# B&R Automation Studio project MotionTestBenchMaster (part 14)

### HMI_ICO.typ
```iecst
TYPE
	HMI_ICO_Type : 	STRUCT
		NextRecipeId : UDINT; (*ID of the next recipe requested from HLI*)
		ActualRecipeId : UDINT; (*ID of the actual recipe*)
		NextRecipeLoadingReq : BOOL; (*Request to download the new recipe*)
		RecipeLoaded : BOOL; (*New recipe downloaded*)
	END_STRUCT;
END_TYPE
```

### HMI_ITC.typ
```iecst
TYPE
	HMI_MachineComm_Type : 	STRUCT
		CapFault : BOOL; (*V4.A.A.1.6.12*)
		SkidFault : BOOL;
		FmcFault : BOOL;
	END_STRUCT;
END_TYPE
```

### HMI_MAU.typ
```iecst
(*DBA glass Status*)

TYPE
	HMI_DMC_Status : 	STRUCT
		Sector1Position : USINT;
		Sector1PistonDown : USINT;
		Sector1RotationToProd : USINT;
		Sector1RotationToCip : USINT;
		Sector1PistonUp : USINT;
		Sector2Position : USINT;
		Sector2PistonDown : USINT;
		Sector2RotationToProd : USINT;
		Sector2RotationToCip : USINT;
		Sector2PistonUp : USINT;
	END_STRUCT;
END_TYPE

(*COMMON*)

TYPE
	HMI_UV_Lamp_Type : 	STRUCT
		ConfigPresent : USINT;
		On : USINT;
		Ready : USINT;
		Alarm : USINT;
	END_STRUCT;
END_TYPE

(*GREASING*)

TYPE
	HMI_GrLb_Data_Type : 	STRUCT
		Alarm : BOOL;
		Pause : UINT; (*[laps]*)
		CycleTimeOut : UINT; (*[s]*)
		CycleNr : UINT; (*[#]*)
	END_STRUCT;
END_TYPE

(*SAFE LOGIC*)

TYPE
	HMI_SL_Info_Type : 	STRUCT
		RemoteCtrlStatus : UINT;
		CRC : UDINT;
		Password : ARRAY[0..15]OF USINT;
		Date : STRING[15];
		Author : STRING[32];
		IDMissed : STRING[80];
		IDMismatches : STRING[80];
		IDDiffFirmware : STRING[80];
		Led : HMI_SL_Led_Type;
	END_STRUCT;
	HMI_SL_Led_Type : 	STRUCT
		FAIL : USINT;
		FW_ACKN : USINT;
		MXCHG : USINT;
		RE : USINT;
	END_STRUCT;
	HMI_SL_PB_Type : 	STRUCT
		Ack_SK : PB_Type;
		Ack1UdId : PB_Type;
		Ack2UdId : PB_Type;
		Ack3UdId : PB_Type;
		Ack4UdId : PB_Type;
		AckMore4UdId : PB_Type;
		AckFW : PB_Type;
		LedTest : PB_Type;
		Scan : PB_Type;
	END_STRUCT;
	HMI_MAU_ChlRns_Type : 	STRUCT  (*master nuovo*)
		AVE260_PauseTimeWithBottles : UINT;
		AVE260_WorkTimeWithBottles : UINT;
		AVE260_PauseTimeWithoutBottles : UINT;
		AVE260_WorkTimeWithoutBottles : UINT;
		AVE261_PauseTimeWithoutBottles : UINT;
		AVE261_WorkTimeWithoutBottles : UINT;
		PauseTimeMaxWithoutChlRns : UINT;
		WorkTimeMaxWithoutChlRns : UINT;
	END_STRUCT;
END_TYPE
```

### HMI_MC.typ
```iecst
TYPE
	ST_HmiNewAxisData : 	STRUCT  (*V4.A.A.1.7.0*)
		rTorque : REAL;
		rTotalPhasingOffset : REAL;
		rMaxTorque : REAL;
		rPosition : REAL;
		rPosition_mm : REAL;
		rVelocity : REAL;
		rMotorTemperature : REAL;
		rLagError : REAL;
		rEncoderTemperature : REAL;
		rSwitchValue : REAL;
		rPrevAx_Position_mm : REAL;
		rHomingOffset : REAL; (*mm*)
		rNextAx_Position_mm : REAL;
		usiHmiName : USINT;
		uiDiagCode : UINT;
		uiAxisID : UINT; (*//Hmi Test*)
		iPrevAx_Number : INT;
		iNextAx_Number : INT;
		xMotorWithBrake : BOOL;
		xVelocityControl : BOOL;
		xInduction : BOOL;
		xReal : BOOL;
		xInitialized : BOOL;
		xEnabled : BOOL;
		xPowered : BOOL;
		xHomed : BOOL;
		xActive : BOOL;
		xInPosition : BOOL;
		xRunning : BOOL;
		xSynchro : BOOL;
		xBrakeReleased : BOOL;
		xFollowingError : BOOL;
		xInError : BOOL;
		xTorqueError : BOOL;
		xThirdPartMotor : BOOL;
		xHmiPresent : BOOL; (*//Hmi Test*)
		xHmiWait : BOOL;
	END_STRUCT;
	ST_HmiAxisData : 	STRUCT
		rTorque : REAL;
		rTotalPhasingOffset : REAL;
		rMaxTorque : REAL;
		rPosition : REAL;
		rPosition_mm : REAL;
		rVelocity : REAL;
		rMotorTemperature : REAL;
		rLagError : REAL;
		rEncoderTemperature : REAL;
		rSwitchValue : REAL;
		rPrevAx_Position_mm : REAL;
		rHomingOffset : REAL; (*mm*)
		rNextAx_Position_mm : REAL;
		usiHmiName : USINT;
		uiDiagCode : UINT;
		iPrevAx_Number : INT;
		iNextAx_Number : INT;
		xMotorWithBrake : BOOL;
		xVelocityControl : BOOL;
		xInduction : BOOL;
		xReal : BOOL;
		xInitialized : BOOL;
		xEnabled : BOOL;
		xPowered : BOOL;
		xHomed : BOOL;
		xActive : BOOL;
		xInPosition : BOOL;
		xRunning : BOOL;
		xSynchro : BOOL;
		xBrakeReleased : BOOL;
		xFollowingError : BOOL;
		xInError : BOOL;
		xTorqueError : BOOL;
		xThirdPartMotor : BOOL;
		xHmiWait : BOOL;
	END_STRUCT;
	ST_HmiMachineStatus : 	STRUCT
		xNoOperationActive : BOOL;
		xAuto : BOOL;
		xAutoCombi : BOOL;
		xPositioning : BOOL;
		xJogMachine : BOOL;
		xBrakeRelease : BOOL;
		xStepByStep : BOOL;
		xEndlessFeed : BOOL;
		xSplittedModality : BOOL;
		xFillerJogStandAlone : BOOL;
		xOutletJogStandAlone : BOOL;
		xInletJogStandAlone : BOOL;
		xFillerStepByStep : BOOL;
		xOutletStepByStep : BOOL;
		xInletStepByStep : BOOL;
		xFillerSlowMotion : BOOL;
		xOutletSlowMotion : BOOL;
		xInletSlowMotion : BOOL;
		xMachineStart : BOOL;
		xMachineSincroStop : BOOL;
		xMachineFixedSpeed : BOOL;
		xMachineSincro : BOOL;
		xMachineSincroInProgress : BOOL;
		xMachineOnError : BOOL;
		xMachineHomed : BOOL;
		xMachineRunning : BOOL;
		rEncoderPosition : REAL;
		rMachineStep : REAL;
	END_STRUCT;
	ST_HmiAxisPresent : 	STRUCT
		_99 : UINT;
		_100 : UINT;
		_105 : UINT;
		_106 : UINT;
		_107 : UINT;
		_108 : UINT;
		_109 : UINT;
		_110 : UINT;
		_111 : UINT;
		_112 : UINT;
		_113 : UINT;
		_114 : UINT;
		_115 : UINT;
		_116 : UINT;
		_117 : UINT;
		_118 : UINT;
		_119 : UINT;
		_120 : UINT;
		_121 : UINT;
		_200 : UINT;
		_211 : UINT;
		_212 : UINT;
		_213 : UINT;
		_214 : UINT;
		_215 : UINT;
		_216 : UINT;
		_217 : UINT;
		_218 : UINT;
		_219 : UINT;
		_300 : UINT;
		_311 : UINT;
		_312 : UINT;
		_313 : UINT;
		_314 : UINT;
		_315 : UINT;
		_316 : UINT;
		_317 : UINT;
		_318 : UINT;
		_319 : UINT;
	END_STRUCT;
	ST_HMIEncoderDiagnostic : 	STRUCT
		Present : BOOL;
		ModuleOK : BOOL;
		Value : DINT;
	END_STRUCT;
END_TYPE
```

### HMI_MNM.typ
```iecst
TYPE
	HMI_SpeedWidget_Type : 	STRUCT
		Modality : BOOL; (*0 = Auto / 1 = Jog*)
		Visibility : BOOL; (*0 = Hidden (Combi Mode) / 1 = Visible*)
		ActualSpeed : DINT; (*Actual Machine Speed [cph]*)
		AutoSpeedReq : DINT; (*Automatic Speed Required (Standalone) [cph]*)
		JogSpeedReq : DINT; (*Jog Speed Required (Standalone) [cph]*)
		Status : USINT; (*0: Error
1: Automatic
2: Jog
3: Adjustement
4: Slow motion forward
5: Slow motion backward*)
	END_STRUCT;
END_TYPE
```

### HMI_MNT.typ
```iecst
TYPE
	HMI_MNT_Type : 	STRUCT
		Macao : HMI_Macao_Type;
		Tpm : ARRAY[0..12]OF HMI_Tpm_Type; (*//v1.5*)
		_201QTB : HMI_Tpm_Type; (*V1.7.4*)
		_202QTB : HMI_Tpm_Type; (*V1.7.4*)
	END_STRUCT;
	HMI_Macao_Type : 	STRUCT
		Counter : ARRAY[0..15]OF UDINT;
		Event : ARRAY[0..7]OF BOOL;
	END_STRUCT;
	HMI_Tpm_Type : 	STRUCT  (*//v1.5*)
		Config : BOOL;
		AnalogNomValueVisible : BOOL;
		AnalogAlarmValueVisible : BOOL; (*V1.7.4*)
		InstrumentFault : BOOL; (*V1.7.4*)
		HmiID : UINT;
		AnalogActValue : REAL;
		AnalogMaxValue : REAL;
		AnalogMinValue : REAL;
		AnalogNomValue : REAL;
		AnalogAlarmValue : REAL; (*V1.7.4*)
	END_STRUCT;
END_TYPE
```

### HMI_OPS.typ
```iecst
TYPE
	HMI_OPS_Zone_Type : 	STRUCT
		Closed : BOOL;
		Locked : BOOL;
		LockSafety : BOOL;
		ShortSafety : BOOL;
		UnlockCommand : BOOL;
		Unlocked : BOOL;
		UnlockEnable : BOOL;
		UnlockRequest : BOOL;
		UnlockSafety : BOOL;
	END_STRUCT;
	HMI_OPS_Door_Type : 	STRUCT
		Confirm : BOOL;
		Lock1oo2 : BOOL;
		LockSafety : BOOL;
		Opened : BOOL;
		ShortCircuit : BOOL;
		UnLock : BOOL;
	END_STRUCT;
	HMI_OPS_Emergency_Type : 	STRUCT
		I_Pressed : BOOL;
		I_short_Fault : BOOL;
	END_STRUCT;
	HMI_OPS_Jog_Type : 	STRUCT
		ShCircPlug : BOOL;
		ShCircStop : BOOL;
		Stop : BOOL;
		Plugged : BOOL;
	END_STRUCT;
	HMI_SafetyWidget_Type : 	STRUCT
		ZoneAlarm : ARRAY[MIN_CFG_SafetyZone..MAX_CFG_SafetyZone]OF BOOL;
		BufferAlarm : BOOL;
	END_STRUCT;
	HMI_OPS_Pictogram_Type : 	STRUCT
		AccesOk : BOOL;
		AccesReq : BOOL;
		Acces : BOOL;
		Chemical : BOOL;
		Temperature : BOOL;
	END_STRUCT;
	HMI_OPS_RfidAccess_Type : 	STRUCT
		Present : BOOL; (*Module Present*)
		CodeFault : BOOL; (*Code discrepancy*)
		KeyFault : BOOL; (*Key not recognised*)
		KeyOk : BOOL; (*Key present and recognised*)
	END_STRUCT;
	HMI_OPS_SafetySwitch_Type : 	STRUCT  (*V4.A.A.1.7.1*) (* *) (*139*)
		ShortFault : BOOL; (*Short circuit fault on PB*) (* *) (*141*)
		SwitchOn : BOOL; (*Switch active*) (* *) (*143*)
		Visibility : BOOL; (*Switch present*) (* *) (*144*)
	END_STRUCT;
END_TYPE
```

### HMI_RNS.typ
```iecst
TYPE
	HMI_RNS_ManualCapsSelection_Type : 	STRUCT  (*V4.A.A.1.7.0*)
		Value : USINT;
		Visibility : BOOL;
	END_STRUCT;
	HMI_RNS_State_Type : 	STRUCT (*V4.A.A.1.7.4*)
		Sequencer : Seq_Type; (*Step Actual*)
		Signals : Signals_Type;
	END_STRUCT;
END_TYPE
```

### HMI_SFT.typ
```iecst
TYPE
	StepAcquisition_Type : 	STRUCT
		Step : USINT;
		_207DSF : StepAcquisition_Sensor_Type;
		_208DSF : StepAcquisition_Sensor_Type;
		_202DSF : StepAcquisition_Sensor_Type;
		_203DSF : StepAcquisition_Sensor_Type;
	END_STRUCT;
	StepAcquisition_Sensor_Type : 	STRUCT
		Visibility : BOOL;
		Value : UINT;
	END_STRUCT;
	MainCounters_Type : 	STRUCT
		PbResetMachineCounters : PB_Type;
		MachineCounters : MachineCounters_Type;
		PbResetCycleCounters : PB_Type;
		CycleCounters : TankCounters_Type;
		PbResetContainersCounters : PB_Type;
		ContainersCounters : ContainersCounters_Type;
		PbResetEcoEitCounters : PB_Type;
		EcoEitCounters : EcoEitCounters_Type;
	END_STRUCT;
	MachineCounters_Type : 	STRUCT
		CapLaps : UDINT; (*Capper torret laps counter*)
		FlrLaps : UDINT; (*Filler laps counter*)
		RnsLaps : UDINT; (*Rinser laps counter*)
		PowerOnCycles : UDINT;
		PowerOnTime : CounterTime_Type;
		RotationTime : CounterTime_Type; (*Machine running hours counter*)
		StartTime : CounterTime_Type;
	END_STRUCT;
	ContainersCounters_Type : 	STRUCT
		CapFault : UDINT;
		FlrBurst : UDINT;
		RnsFault : UDINT;
		FlrFault : UDINT;
		Ejected : UDINT;
		Entered : UDINT;
		Produced : UDINT;
		StartTime : CounterTime_Type;
	END_STRUCT;
	TankCounters_Type : 	STRUCT
		ProductionCounter : UDINT;
		ProductionTime : CounterTime_Type;
		CipCounter : UDINT;
		CipTime : CounterTime_Type;
		StartTime : CounterTime_Type;
	END_STRUCT;
	EcoEitCounters_Type : 	STRUCT
		ElectricalPowerKWH : REAL; (*[KWH]*)
		ElectricalPowerKVAR : REAL; (*[KVAR]*)
		StartTime : CounterTime_Type;
	END_STRUCT;
	HmiCounterData_Type : 	STRUCT
		Description : STRING[25];
		Unit : STRING[8];
		PbReset : PB_Type;
		ConfigPresent : BOOL;
		ValuePresent : BOOL;
		TimePresent : BOOL;
		StartDatePresent : BOOL;
	END_STRUCT;
	CounterCfg_Type : 	STRUCT
		MachineCounters : MachineCountersCfg_Type;
		ContainersCounters : ContainersCountersCfg_Type;
		ProcessCounters : ProcessCountersCfg_Type;
		EcoCounters : EcoCountersCfg_Type;
	END_STRUCT;
	CounterData_Type : 	STRUCT
		MachineCounters : MachineCountersData_Type;
		ContainersCounters : ContainersCountersData_Type;
		ProcessCounters : ProcessCountersData_Type;
		EcoCounters : EcoCountersData_Type;
	END_STRUCT;
	HMI_CounterPage_Type : 	STRUCT
		Partial : HMI_CounterPage2_Type;
		Total : HMI_CounterPage2_Type;
	END_STRUCT;
	HMI_CounterPage2_Type : 	STRUCT
		Data : ARRAY[0..15]OF HmiCounterData_Type;
		Cfg : ARRAY[0..15]OF Counters_Type;
	END_STRUCT;
END_TYPE

(*Machine Counter*)

TYPE
	MachineCountersCfg_Type : 	STRUCT
		HmiData : ARRAY[0..15]OF HmiCounterData_Type;
	END_STRUCT;
	MachineCountersData_Type : 	STRUCT
		CounterData : ARRAY[0..15]OF Counters_Type;
	END_STRUCT;
END_TYPE

(*Containers Counter*)

TYPE
	ContainersCountersCfg_Type : 	STRUCT
		HmiData : ARRAY[0..15]OF HmiCounterData_Type;
	END_STRUCT;
	ContainersCountersData_Type : 	STRUCT
		CounterData : ARRAY[0..15]OF Counters_Type;
	END_STRUCT;
END_TYPE

(*Process Coutner*)

TYPE
	ProcessCountersCfg_Type : 	STRUCT
		HmiData : ARRAY[0..15]OF HmiCounterData_Type;
	END_STRUCT;
	ProcessCountersData_Type : 	STRUCT
		CounterData : ARRAY[0..15]OF Counters_Type;
	END_STRUCT;
END_TYPE

(*Eco Counter*)

TYPE
	EcoCountersCfg_Type : 	STRUCT
		HmiData : ARRAY[0..15]OF HmiCounterData_Type;
	END_STRUCT;
	EcoCountersData_Type : 	STRUCT
		CounterData : ARRAY[0..15]OF Counters_Type;
	END_STRUCT;
END_TYPE

(*FILLING VALVE*)

TYPE
	DummyContainerDataStructure_Type : 	STRUCT
		FillingNozzle : USINT;
		DummyInstalled : BOOL; (*SHIFT master nuovo*)
		DummyNotInserted : BOOL;
		DummyRemoved : BOOL;
		DummyNotRemoved : BOOL;
	END_STRUCT;
	FillingValveDataStructure_Type : 	STRUCT
		FillingDisabled : BOOL; (*SHIFT master nuovo*)
		ContainerBurst : BOOL;
		ContainerPresence : BOOL;
		PreClosingEnd : BOOL;
		WashingLapsEnd : BOOL;
		PreClosingCmdLap1 : BOOL;
		PreClosingCmdLap2 : BOOL;
		PreClosingCmdLap3 : BOOL;
		PreClosingCmdLap4 : BOOL;
		PreClosingCmdLap5 : BOOL;
		PreClosingCmdLap6 : BOOL;
		PreClosingCmdLap7 : BOOL;
		OperatorInspectionReq : BOOL;
		PreClosingActualLap : USINT;
		WashingLaps : USINT;
		ConsecutiveFillNotOk : USINT;
		AbsoluteFillNotOk : USINT;
		ConsecutiveBurst : USINT;
		AbsoluteBurst : USINT;
	END_STRUCT;
	HMI_SFT_BurstData_Type : 	STRUCT
		ColorStatus : USINT;
		Counter : UINT;
	END_STRUCT;
END_TYPE

(*Sampling*)

TYPE
	HMI_SFT_SamplingMold_Type : 	STRUCT  (*V1.61*)
		Present : BOOL;
		Selected : BOOL;
	END_STRUCT;
END_TYPE
```

### HMI.typ
```iecst
TYPE
	Step_Type : 	STRUCT
		Config_Visualization : BOOL;
		Preset : REAL; (*Preset Step Time*)
		Actual : REAL; (*Actual Step Time*)
		StepIndex : UINT; (*Actual Sequencer Step Number*)
		StepIndexText : UINT; (*Request Step Text to HMI*)
	END_STRUCT;
	Signals_Type : 	STRUCT
		DigitalIn : ARRAY[1..5]OF HMI_DigitalITC_Type;
		AnalogIn : ARRAY[1..2]OF HMI_AnalogITC_Type;
		DigitalOut : ARRAY[1..5]OF HMI_DigitalITC_Type;
		AnalogOut : ARRAY[1..2]OF HMI_AnalogITC_Type;
	END_STRUCT;
	Seq_Type : 	STRUCT
		TextBar : ARRAY[0..4]OF SeqTextBar_Type;(*master nuovo*)
		InfoBox : ARRAY[0..5]OF SeqInfo_Type; (*Preset Step Time*)
	END_STRUCT;
	SeqTextBar_Type : 	STRUCT
		Visibility : BOOL;
		IndexNr : UINT; (*Actual Sequencer Step Number*)
		IndexText : UINT; (*Request Step Text to HMI*)
	END_STRUCT;
	SeqInfo_Type : 	STRUCT
		Visibility : BOOL;
		IndexText : STRING[20]; (*Request Step Text to HMI*)
		Unit : UINT;
		ProgressVisibility : BOOL; (*Step Progress Visibility*)
		Progress : REAL; (*Step Progress Time*)
		Preset : REAL; (*Preset Step Time*)
		Actual : REAL; (*Actual Step Time*)
	END_STRUCT;
	Info_Type : 	STRUCT  (*v1.4*)
		Visibility : BOOL;
		Preset : REAL; (*Preset Value*)
		Actual : REAL; (*Actual value*)
	END_STRUCT;
	Data_Type : 	STRUCT  (*v1.7.4a*)
		Visibility : BOOL;
		StringLineNameVisibility : BOOL; (*0=Fix text displayed-1= String displayed*)
		DataValueVisibility : BOOL; (*0=String displayed-1= Numeric value displayed*)
		LineName : STRING[100]; (*Line Name*)
		DataText : STRING[100]; (*Data Text in Case of String*)
		DataValue : REAL; (*Data Value in Case of Numeric*)
	END_STRUCT;
	HMI_CounterHome_Type : 	STRUCT  (*V4.A.A.1.6.8*)
		SS2P : SS2P_Type;
		CounterValue : ARRAY[0..1]OF UDINT;
	END_STRUCT;
END_TYPE
```

### HMI_BTC.typ - not listed in the package file held
```iecst
(*BOTTLE BOTTOM COOLING*)

TYPE
	HMI_BTC_State_Type : 	STRUCT
		Sequencer : Seq_Type; (*Step Actual*)
		Signals : Signals_Type;
	END_STRUCT;
END_TYPE
```

### Package Logical/02_HMI/HMI_Variables - HMI Global variables

### HMI_AID.var
```iecst
VAR
	HMI_CmdBar_PB : ARRAY[MIN_CmdBar_PB..MAX_CmdBar_PB] OF CmdBarPB_Type := [25((Enable:=FALSE,LampON:=FALSE,Blink:=FALSE,Visibility:=FALSE,ON:=FALSE,Command:=FALSE))]; (*1: Mixer Start/Stop
2: Filler Start/Stop
3: Labeller Start/Stop
4: Blower Start/Stop
5: Labeller Master/Slave
6: Preform Loading
7: Bottle with label ejection
8: Empty bottle ejection
9: Preform ejection
10: Filler/Labeller coupling
11: Labeller/Blower coupling
12: Filler door unlock
13: Labeller door unlock
14: Blower door unlock*)
	HMI_PB : ARRAY[MIN_PB_CFG..MAX_PB_CFG] OF PB_Type;
	HMI_SS2P : ARRAY[MIN_SS2P_CFG..MAX_SS2P_CFG] OF SS2P_Type;
	HMI_SS2P_Custom : ARRAY[0..2] OF SS2PCustom_Type; (*V4.A.A.1.6.13*)
END_VAR
```

### HMI_ALR.var
```iecst
VAR
	HMI_ALR : ARRAY[1..8000] OF BYTE;
	HMI_MSG : ARRAY[1..2000] OF BOOL;
END_VAR
```

### HMI_CAP.var
```iecst
VAR
	HMI_CAP_Step : INT;
	HMI_CAP_PB : ARRAY[MIN_PB_CFG..MAX_PB_CFG] OF PB_Type;
	HMI_CAP_SS2P : ARRAY[MIN_SS2P_CFG..MAX_SS2P_CFG] OF SS2P_Type;
	HMI_CAP_SS3P : ARRAY[MIN_SS3P_CFG..MAX_SS3P_CFG] OF SS3P_Type;
	HMI_CAP_CapsTypeCFG : STRING[500];
	HMI_CAP_ManualCapsSelection : HMI_CAP_ManualCapsSelection_Type;
	HMI_CAP_State : HMI_CAP_State_Type;
	HMI_CAP_ConfigStructure : HMI_CAP_ConfigStructure_Type;
	HMI_CAP_BufferPresent : BOOL; (*Buffer Present bit for HMI*)
	HMI_CAP_MultiChoiceMng : USINT; (*1=Arol Equatorque ; 2=Arol Equatorque\Multybody ; 3=Zalkin Brushless ; 4=Siko Multybody*)
	HMI_CAP_Brush : HMI_CAP_Brush_Type; (*Capper Brushless Arol/Zalkin v1.4*)
	HMI_CAP_DataCfg : ARRAY[1..10] OF HMI_COP_ZoneCfg_Type; (*Column Configuration Capper Brushless Arol/Zalkin v1.4*)
	HMI_CAP_BufferAdjust : Info_Type; (*//V4.A.A.1.6.11*)
	HMI_CAP_HRM : HMI_CAP_HRM_Type; (*//V4.A.A.1.6.11*)
END_VAR
(*GREASING*)
VAR
	HMI_CAP_GreasingState : Seq_Type;
	HMI_CAP_GreasingState2 : Seq_Type; (*//V4.A.A.1.6.11*)
	HMI_CAP_GreasingData2 : HMI_CAP_Greasing_Type; (*//V4.A.A.1.6.11*)
	HMI_CAP_GreasingData : HMI_CAP_Greasing_Type;
END_VAR
(*MOTORS*)
VAR
	HMI_202GPE : HMI_GreasingPump_Type;
	HMI_203GPE : HMI_GreasingPump_Type; (*//V4.A.A.1.6.11*)
	HMI_206MMR : HMI_Motor_FC_Type; (*Head rotation motor*)
	HMI_206MMRBrake : HMI_Motor_Type; (*Head rotation motor*)
	HMI_207MMR : HMI_Motor_FC_Type; (*Hopper motor chute 1*)
	HMI_230MMR : HMI_Motor_Type; (*Dust removal motor on caps channel*)
	HMI_231MMR : HMI_Motor_Type; (*Dust removal motor on buffer //V4.A.A.1.6.11*)
	HMI_229MMR : HMI_Motor_Type; (*Adjustment panel motor //V4.A.A.1.6.11*)
	HMI_212MMR : HMI_Motor_FC_Type; (*Buffer rotation motor*)
	HMI_213MMR : HMI_Motor_Type; (*Head rotation motor fun*)
	HMI_214MMR : HMI_Motor_FC_Type; (*Hopper motor chute 2*)
	HMI_215MMR : HMI_Motor_FC_Type; (*Hopper motor chute 3*)
END_VAR
(*IONIZER*)
VAR
	HMI_201DRC_SwitchFeedback : HMI_DI_Type;
	HMI_201DRC : HMI_Motor_Type; (*Ionizer*)
END_VAR
(*UV LAMP*)
VAR
	HMI_201LLC : HMI_Motor_Type; (*UV lamp Chute 1*)
	HMI_202LLC : HMI_Motor_Type; (*UV lamp Chute 2*)
	HMI_203LLC : HMI_Motor_Type; (*UV lamp Chute 3*)
END_VAR
(*SIKO MULTIBODY V1.61*)
VAR
	HMI_CAP_SikoMotorSetPointEnable : BOOL; (*Multibody Siko Motor for Automatic Change Capper Guide Enable Set Point For Calibration*)
	HMI_CAP_SikoMotor : ARRAY[0..5] OF HMI_CAP_SikoMotor_Type; (*Multibody Siko Motor for Automatic Change Capper Guide *)
END_VAR
(*DRIVERS*)
VAR
	HMI_VFD_206MMR : HMI_Danfoss_Diag_Type; (*Head rotation motor*)
	HMI_VFD_207MMR : HMI_Danfoss_Diag_Type; (*Hopper motor chute 1*)
	HMI_VFD_230MMR : HMI_Danfoss_Diag_Type; (*Dust remover motor*)
	HMI_VFD_212MMR : HMI_Danfoss_Diag_Type; (*Buffer rotation motor*)
	HMI_VFD_213MMR : HMI_Danfoss_Diag_Type; (*Head rotation motor fun*)
	HMI_VFD_214MMR : HMI_Danfoss_Diag_Type; (*Hopper motor chute 2*)
	HMI_VFD_215MMR : HMI_Danfoss_Diag_Type; (*Hopper motor chute 3*)
	HMI_ST3B : HMI_Analog_IN_Type; (*Tempaerature sensor Equatorque motor//V4.A.A.1.6.12*)
	HMI_ST3A : HMI_Analog_IN_Type; (*Tempaerature sensor Equatorque motor//V4.A.A.1.6.12*)
END_VAR
(*VALVES*)
VAR
	HMI_201CPC : HMI_Valve_Type; (*EV chute 1 caps release*)
	HMI_202CPC : HMI_Valve_Type; (*EV chute 2 caps release*)
	HMI_205CPC : HMI_Valve_Type; (*EV caps block chute 1*)
	HMI_206CPC : HMI_Valve_Type; (*EV caps block chute 2*)
	HMI_207CPC : HMI_Valve_Type; (*EV cap discharge door*)
	HMI_212CPC : HMI_Valve_Type; (*EV open buffer discharge door*)
	HMI_213CPC : HMI_Valve_Type; (*EV buffer lifting*)
	HMI_214CPC : HMI_Valve_Type; (*EV buffer lock*)
	HMI_215CPC : HMI_Valve_Type; (*EV lock size change guide*)
	HMI_216CPC : HMI_Valve_Type; (*EV 3 size change guide*)
	HMI_217CPC : HMI_Valve_Type; (*EV 4 size change guide*)
	HMI_218CPC : HMI_Valve_Type; (*EV sport size change guide*)
	HMI_219CPC : HMI_Valve_Type; (*EV open channel discharge door*)
	HMI_220CPC : HMI_Valve_Type; (*FREE v1.7.6*)
	HMI_221CPC : HMI_Valve_Type; (*EV chute 3 caps release*)
	HMI_222CPC : HMI_Valve_Type; (*EV caps block chute 3*)
	HMI_223CPC : HMI_Valve_Type; (*EV buffer vibrator*)
	HMI_224CPC : HMI_Valve_Type; (*EV cam position*)
	HMI_225CPC : HMI_Valve_Type; (*EV cam locking*)
	HMI_226CPC : HMI_Valve_Type; (*EV opening door UV Lamp A V. 1.1*)
	HMI_227CPC : HMI_Valve_Type; (*EV  Block Caps Outlet Chute 1*)
	HMI_228CPC : HMI_Valve_Type; (*EV transfer Starwheel air soleniod valve DA VERIFICARE*)
	HMI_229CPC : HMI_Valve_Type; (*EV transfer Starwheel air soleniod valve DA VERIFICARE*)
	HMI_232CPC : HMI_Valve_Type; (*EV opening door UV Lamp B V. 1.1*)
	HMI_233CPC : HMI_Valve_Type;
	HMI_234CPC : HMI_Valve_Type; (*EV Caps Ejection Cap Feeder V4.A.A.1.6.12*)
	HMI_235CPC : HMI_Valve_Type; (*v1.7.4*)
	HMI_236CPC : HMI_Valve_Type; (*v1.7.4*)
	HMI_237CPC : HMI_Valve_Type; (*v1.7.4*)
	HMI_238CPC : HMI_Valve_Type; (*v1.7.4*)
	HMI_201EVC : HMI_Valve_Type; (*Air blowing for cap release 1 V1.6*)
	HMI_203EVC : HMI_Valve_Type; (*Air blowing for cap release 2 V1.6*)
	HMI_207EVC : HMI_Valve_Type; (*Air blowing for cap release 3 V1.6*)
	HMI_209EVC : HMI_Valve_Type; (*v1.7.4*)
	HMI_210EVC : HMI_Valve_Type; (*Air blowing for buffer emptying*)
	HMI_211EVC : HMI_Valve_Type; (*Buffer air blowing for caps release*)
	HMI_212EVC : HMI_Valve_Type; (*Air blowing for chute emptying*)
	HMI_213EVC : HMI_Valve_Type; (*Air blowing caps ionizer chute 1*)
	HMI_214EVC : HMI_Valve_Type; (*Air blowing caps ionizer chute 2*)
	HMI_215EVC : HMI_Valve_Type; (*Air blowing caps ionizer chute 3*)
	HMI_216EVC : HMI_Valve_Type; (*Air blowing for chute emptying by pep*)
	HMI_227EVC : HMI_Valve_Type; (*v1.7.4*)
	HMI_228EVC : HMI_Valve_Type; (*v1.7.4*)
	HMI_229EVC : HMI_Valve_Type; (*v1.7.4*)
	HMI_203EVF : HMI_Valve_Type; (*Air blowing caps (Drying)*)
	HMI_AVC : ARRAY[MIN_CFG_AVC..MAX_CFG_AVC] OF HMI_Valve_Type; (*Caps Treatment Valves V4.A.A.1.7.4*)
END_VAR
(*SENSOR*)
VAR
	HMI_201DSC : HMI_Photocell_Type; (*Caps/crowns release check*)
	HMI_202DSC : HMI_DI_Type; (*Low level caps/crowns presence chute 1*)
	HMI_204DSC : HMI_DI_Type; (*Head 1 sensor*)
	HMI_205DSC : HMI_DI_Type; (*Lack of caps (Quibuf infeed)*)
	HMI_210DSC : HMI_DI_Type; (*Cap Overturned hight Cap Feeder  V4.A.A.1.7.1*)
	HMI_211DSC : HMI_DI_Type; (*Cap Overturned low  Cap Feeder  V4.A.A.1.7.1*)
	HMI_216DSC : HMI_DI_Type; (*Low level caps/crowns presence chute 2*)
	HMI_217DSC : HMI_DI_Type; (*Low level caps/crowns presence chute 3*)
	HMI_218DSC : HMI_DI_Type; (*Upside down caps check chute 1 high*)
	HMI_219DSC : HMI_DI_Type; (*Upside down caps check chute 1 low*)
	HMI_220DSC : HMI_DI_Type; (*Upside down caps check chute 2 high*)
	HMI_221DSC : HMI_DI_Type; (*Upside down caps check chute 2 low*)
	HMI_222DSC : HMI_DI_Type; (*Upside down caps check chute 3 high*)
	HMI_223DSC : HMI_DI_Type; (*Upside down caps check chute 3 low*)
	HMI_224DSC : HMI_DI_Type; (*Ionizer pressure switch chute 1*)
	HMI_225DSC : HMI_DI_Type; (*Ionizer pressure switch chute 2*)
	HMI_226DSC : HMI_DI_Type; (*Ionizer pressure switch chute 3*)
	HMI_227DSC : HMI_DI_Type; (*Lubrication door sensor*)
	HMI_228DSC : HMI_DI_Type; (*Fixed part lubrication check*)
	HMI_229DSC : HMI_DI_Type; (*Rotating part lubrication check*)
	HMI_230DSC : HMI_DI_Type; (*Lubrication pipe inserted sensor*)
	HMI_231DSC : HMI_DI_Type; (*Turret cam position analog sensor*)
	HMI_232DSC : HMI_DI_Type; (*Caps buffer full*)
	HMI_233DSC : HMI_DI_Type; (*Caps channel discharge gate sensor*)
	HMI_234DSC : HMI_DI_Type; (*Lubrication phase sensor*)
	HMI_235DSC : HMI_DI_Type; (*Buffer in high position*)
	HMI_236DSC : HMI_DI_Type; (*Buffer in low position*)
	HMI_237DSC : HMI_DI_Type; (*Buffer lock inserted*)
	HMI_238DSC : HMI_DI_Type; (*Caps buffer max level chute 1*)
	HMI_239DSC : HMI_DI_Type; (*Caps buffer max level chute 2*)
	HMI_240DSC : HMI_DI_Type; (*Caps buffer max level chute 3*)
	HMI_241DSC : HMI_DI_Type; (*Hopper level chute 1*)
	HMI_242DSC : HMI_DI_Type; (*Hopper level chute 2*)
	HMI_243DSC : HMI_DI_Type; (*Hopper level chute 3*)
	HMI_244DSC : HMI_DI_Type; (*Max level caps/crowns chute 1*)
	HMI_245DSC : HMI_DI_Type; (*Max level caps/crowns chute 2*)
	HMI_246DSC : HMI_DI_Type; (*Max level caps/crowns chute 3*)
	HMI_247DSC : HMI_DI_Type; (*Medium level caps/crowns chute 1*)
	HMI_248DSC : HMI_DI_Type; (*Medium level caps/crowns chute 2*)
	HMI_249DSC : HMI_DI_Type; (*Medium level caps/crowns chute 3*)
	HMI_250DSC : HMI_DI_Type; (*Side door hopper sport*)
	HMI_251DSC : HMI_DI_Type; (*Top door hopper sport*)
	HMI_252DSC : HMI_DI_Type; (*Uv lamp door*)
	HMI_253DSC : HMI_DI_Type; (*Sensore carter posteriore*)
	HMI_254DSC : HMI_DI_Type; (*Sensore di fase per lubrificazione*)
	HMI_255DSC : HMI_DI_Type; (*Sensore di lubrificazione della parte fissa*)
	HMI_256DSC : HMI_DI_Type; (*Sensore di lubrificazione della parte rotante*)
	HMI_257DSC : HMI_DI_Type; (*Sensore di inserimento del raccordo di lubrificazione della parte rotante *)
	HMI_258DSC : HMI_DI_Type; (*Sensore carter superiore  //V4.A.A.1.6.11*)
	HMI_259DSC : HMI_DI_Type; (*Sensore di lubrificazione rotazione teste  //V4.A.A.1.6.11*)
	HMI_260DSC : HMI_DI_Type; (*Sensore di inserimento del raccordo di lubrificazione della parte rotante riduttore rotazione teste  //V4.A.A.1.6.11*)
	HMI_261DSC : HMI_DI_Type; (*Sensore limite minimo posizione pannello //V4.A.A.1.6.11*)
	HMI_262DSC : HMI_DI_Type; (*Sensore zero encoder //V4.A.A.1.6.11*)
	HMI_263DSC : HMI_DI_Type; (*Sensore limite massimo posizione pannello //V4.A.A.1.6.11*)
	HMI_264DSC : HMI_Photocell_Type; (*Caps/Crown release check on bottle//V4.A.A.1.6.12h*)
	HMI_266DSC : HMI_DI_Type; (*v1.7.4*)
	HMI_267DSC : HMI_DI_Type; (*v1.7.5*)
	HMI_268DSC : HMI_DI_Type; (*v1.7.5*)
	HMI_270DSC : HMI_DI_Type; (*Caps Belt Sensor  // v1.7.4*)
END_VAR
```

### HMI_RNS.var
```iecst
(*RINSER*)
VAR
	HMI_RNS_PB : ARRAY[MIN_PB_CFG..MAX_PB_CFG] OF PB_Type;
	HMI_RNS_SS2P : ARRAY[MIN_SS2P_CFG..MAX_SS2P_CFG] OF SS2P_Type;
	HMI_RNS_SS3P : ARRAY[MIN_SS3P_CFG..MAX_SS3P_CFG] OF SS3P_Type;
	HMI_RNS_MultiChoiceMng : USINT; (*0=Rinser Instant Data Not Present  1=Rinser Instant Data Present V4.A.A.1.7.0*)
	HMI_RNS_State : HMI_RNS_State_Type;
	HMI_RNS_NozzleData : ARRAY[1..15] OF RNS_NozzleData_Type; (*V4.A.A.1.7.0*)
	HMI_RNS_ManualSelection : HMI_RNS_ManualCapsSelection_Type; (*V4.A.A.1.7.0*)
	HMI_RNS_TypeCFG : STRING[500]; (*V4.A.A.1.7.0*)
	HMI_RNS_Treatments : ARRAY[0..19] OF HMI_ComboBoxElements_Type := [(Present:=TRUE,Name:='Full Treatment'),(Present:=TRUE,Name:='Water Only'),(Present:=TRUE,Name:='Air Only'),14((0)),10((0)),1((0)),2((0))]; (*V4.A.A.1.7.0*)
END_VAR
```

### HMI_CO.var
```iecst
VAR
	HMI_CO_SS2P : ARRAY[MIN_SS2P_CFG..MAX_SS2P_CFG] OF SS2P_Type;
	HMI_APCO_TypeOfChangeCFG : STRING[500];
	HMI_APCO_TypeOfChange : ARRAY[1..16] OF BOOL; (*V4.A.A.1.6.12*)
END_VAR
VAR RETAIN
	HMI_APCO : HMI_APCO_Type;
END_VAR
```

### HMI_COP.var
```iecst
VAR
	HMI_COP_StatusWidget : HMI_COP_StatusWidget_Type;
END_VAR
VAR RETAIN
	HMI_COP_PB : ARRAY[MIN_PB_CFG..MAX_PB_CFG] OF PB_Type;
	HMI_COP_SS2P : ARRAY[MIN_SS2P_CFG..MAX_SS2P_CFG] OF SS2P_Type;
	HMI_COP_SS3P : ARRAY[MIN_SS3P_CFG..MAX_SS3P_CFG] OF SS3P_Type;
END_VAR
VAR
	HMI_COP_RcpTemp : HMI_COP_Rcp_Type;
END_VAR
VAR RETAIN
	HMI_COP_RcpSelection : ARRAY[0..CST_COP_RcpMax] OF HMI_COP_RcpSelection_Type;
END_VAR
VAR
	HMI_COP_RcpInfo : HMI_COP_RcpInfo_Type;
	HMI_COP_ZoneCfg : ARRAY[1..32] OF HMI_COP_ZoneCfg_Type;
END_VAR
VAR RETAIN
	HMI_RCP_COP_Mngt : RCP_Management_Type;
	HMI_COP_Rcp : HMI_COP_Rcp_Type;
END_VAR
VAR
	HMI_COP_State : HMI_COP_State_Type;
	HMI_COP_PhaseTypeCFG : STRING[500];
	HMI_COP_FuTypeCFG : UDINT;
	HMI_COP_FuGunTypeCFG : UDINT;
	HMI_COP_FuDrainableCFG : UDINT;
	HMI_COP_ITC : HMI_COP_ITC_Type;
	HMI_COP_OptPlangerPresent : BOOL; (*vrma*)
END_VAR
VAR RETAIN
	HMI_RCP_COP_SelectedRecipeName : STRING[70]; (*v999hema*)
END_VAR
```

### HMI_CRW.var
```iecst
VAR
	HMI_CRW_Step : INT;
	HMI_CRW_PB : ARRAY[MIN_PB_CFG..MAX_PB_CFG] OF PB_Type;
	HMI_CRW_SS2P : ARRAY[MIN_SS2P_CFG..MAX_SS2P_CFG] OF SS2P_Type;
	HMI_CRW_SS3P : ARRAY[MIN_SS3P_CFG..MAX_SS3P_CFG] OF SS3P_Type;
	HMI_CRW_CrownsTypeCFG : STRING[500];
	HMI_CRW_ManualCapsSelection : HMI_CRW_ManualCrwSelection_Type;
	HMI_CRW_ConfigStructure : HMI_CRW_ConfigStructure_Type;
END_VAR
(*VALVES*)
VAR
	HMI_230CPC : HMI_Valve_Type;
	HMI_231CPC : HMI_Valve_Type; (*EV chute 1 crowns release*)
	HMI_231EVC : HMI_Valve_Type;
	HMI_205EVC : HMI_Valve_Type; (*EXTRACTOR CLEANING BLOWING VALVE vrma*)
	HMI_274DSC : HMI_DI_Type; (*Head 1 sensor*) (*master nuovo*)
END_VAR
```

### HMI_CSR.var
```iecst
VAR
	HMI_CSR_PB : ARRAY[MIN_PB_CFG..MAX_PB_CFG] OF PB_Type;
	HMI_CSR_SS2P : ARRAY[MIN_SS2P_CFG..MAX_SS2P_CFG] OF SS2P_Type;
	HMI_CSR_SS3P : ARRAY[MIN_SS3P_CFG..MAX_SS3P_CFG] OF SS3P_Type;
END_VAR
(*SENSORS*)
VAR
	HMI_LTK : ARRAY[MIN_CFG_LTx..MAX_CFG_LTx] OF HMI_Analog_IN_Type;
END_VAR
(*MOTORS*)
VAR
	HMI_VFD_RnsLift : HMI_Danfoss_Diag_Type; (*master nuovo*)
	HMI_VFD_TnkLift : HMI_Danfoss_Diag_Type; (*master nuovo*)
	HMI_RnsLift : HMI_Motor_FC_Type; (*master nuovo*)
	HMI_TnkLift : HMI_Motor_FC_Type; (*master nuovo*)
	HMI_2768U0 : HMI_Motor_Type;
	HMI_2809M2 : HMI_Motor_Type; (*master nuovo*)
	HMI_2808M1 : HMI_Motor_Type;
	HMI_2806M1 : HMI_Motor_Type;
	HMI_2806M1_Brake : HMI_Motor_Type; (*master nuovo*)
	HMI_CSR_TnkLinftingMotor : HMI_Motor_Type; (*Tank Lift motor*)
END_VAR
(*VALVES*)
VAR
	HMI_204CPC : HMI_Valve_Type;
	HMI_202CPB : HMI_Valve_Type; (*Containers sectors block*)
	HMI_YV26 : HMI_Valve_Type; (*master nuovo*)
	HMI_YV39 : HMI_Valve_Type; (*master nuovo*)
END_VAR
(*Sequencer Step*)
VAR
	HMI_CSR_State : Seq_Type;
	HMI_CSR_Column : ARRAY[1..3] OF HMI_Column_Type;
	HMI_CSR_SCU : HMI_SCU_Type;
	HMI_CSR_Data : HMI_CSR_Data_Type;
	HMI_212DSB : HMI_DI_Type; (*master nuovo*)
	HMI_213DSB : HMI_DI_Type; (*master nuovo*)
	HMI_3565S5 : HMI_DI_Type; (*master nuovo*)
	HMI_3565S7 : HMI_DI_Type; (*master nuovo*)
	HMI_SQ26 : HMI_DI_Type; (*master nuovo*)
	HMI_SQ45A2 : HMI_DI_Type; (*master nuovo*)
	HMI_SQ45A1 : HMI_DI_Type; (*master nuovo*)
	HMI_SQ70 : HMI_DI_Type; (*master nuovo*)
	HMI_SQ5 : HMI_DI_Type; (*master nuovo*)
	HMI_SQ40 : HMI_DI_Type; (*master nuovo*)
	HMI_SQ6 : HMI_DI_Type; (*master nuovo*)
	HMI_CSR_SikoActualPosition : HMI_CSR_SikoActualPosition_Type; (*master nuovo*)
	HMI_CSR_SikoConveyorData : HMI_CSR_SikoMotorData_Type; (*master nuovo*)
	HMI_CSR_SikoGuideData : HMI_CSR_SikoMotorData_Type; (*master nuovo*)
	HMI_238DSE : HMI_DI_Type; (*Belt Lifting Height Sensor*) (*master nuovo*)
	HMI_243DSE : HMI_DI_Type; (*Body Guide Presence*) (*master nuovo*)
END_VAR
```

### HMI_DMC.var
```iecst
VAR
	HMI_DMC_PB : ARRAY[MIN_PB_CFG..MAX_PB_CFG] OF PB_Type;
	HMI_DMC_AutoModeStatus : HMI_DMC_Status;
	HMI_DMC_ManModeStatus : HMI_DMC_Status;
END_VAR
VAR RETAIN
	HMI_DMC_SS2P : ARRAY[MIN_SS2P_CFG..MAX_SS2P_DMC] OF SS2P_Type;
END_VAR
VAR
	HMI_DMC_State : Seq_Type;
	HMI_DMC_Number : UINT;
	HMI_DMC_InsertionSensor : HMI_DI_Type;
	HMI_211EVF : HMI_Valve_Type;
	HMI_210EVF : HMI_Valve_Type;
	HMI_DMC_InsertionPiston : HMI_Valve_Type;
	HMI_DMC_Sector2LastValveNum : INT;
	HMI_DMC_Sector2FirstValveNum : INT;
	HMI_DMC_Sector1LastValveNum : INT;
	HMI_DMC_Installed : BOOL;
	HMI_DMC_Visualization : BOOL;
	HMI_DMC_AbortFromOperatorCheck : BOOL;
	HMI_DMC_OkFromOperatorCheck : BOOL;
	HMI_DMC_TankHeightPosOk : BOOL;
	HMI_DMC_StepActual : USINT;
END_VAR
```

### HMI_CFG.var
```iecst
VAR
	HMI_PAO : HMI_PAO_Type;
	HMI_CFG_Display : ARRAY[1..20] OF HMI_CFG_Display_Type;
	HMI_CFG_Selection : INT;
	HMI_CFG_Reset : BOOL;
END_VAR
```

### HMI_GNS.var
```iecst
VAR
	HMI_204PSF : HMI_DI_Type;
	HMI_204EVF : HMI_Valve_Type;
	HMI_201PTF : HMI_Analog_IN_Type;
	HMI_205PTF : HMI_Analog_IN_Type;
	HMI_206PTF : HMI_Analog_IN_Type;
	HMI_204PTF : HMI_Analog_IN_Type;
	HMI_201QTB : HMI_Analog_IN_Type; (*Basement Air Control - CO2 Sensor //v1.7.4*)
	HMI_201QTB_Warning : HMI_DI_Type; (*Basement Air Control - CO2 Sensor Warning//v1.7.4*)
	HMI_201QTB_Alarm : HMI_DI_Type; (*Basement Air Control - CO2 Sensor //v1.7.4*)
	HMI_201QTE : HMI_Analog_IN_Type; (*Filler Air Control - CO2 Sensor //v1.7.4*)
	HMI_201QTE_Warning : HMI_DI_Type; (*Filler Air Control - CO2 Sensor Warning//v1.7.4*)
	HMI_201QTE_Alarm : HMI_DI_Type; (*Filler Air Control - Ozozne Sensor Alarm//v1.7.4*)
	HMI_202QTB : HMI_Analog_IN_Type; (*Basement Air Control - CO2 Sensor //v1.7.4*)
	HMI_202QTB_Warning : HMI_DI_Type; (*Basement Air Control - Ozozne Sensor Warning//v1.7.4*)
	HMI_202QTB_Alarm : HMI_DI_Type; (*Basement Air Control - Ozozne Sensor Alarm//v1.7.4*)
	HMI_202QTE : HMI_Analog_IN_Type; (*Filler Air Control - Ozozne Sensor Alarm//v1.7.4*)
	HMI_202QTE_Warning : HMI_DI_Type; (*Filler Air Control - Ozozne Sensor Warning//v1.7.4*)
	HMI_202QTE_Alarm : HMI_DI_Type; (*Filler Air Control - Ozozne Sensor Alarm//v1.7.4*)
	HMI_217DSR : HMI_DI_Type; (*V4.A.A.1.6.12h*)
	HMI_296CPB_I : HMI_DI_Type; (*V4.A.A.1.7.0 Rinser Bypass control*)
	HMI_297CPB_I : HMI_DI_Type; (*V4.A.A.1.7.0 Rinser Bypass control*)
	HMI_224DSB : HMI_DI_Type; (*Doser Bypass control*)
	HMI_225DSB : HMI_DI_Type; (*Doser Bypass control*)
	HMI_226DSB : HMI_DI_Type; (*Doser Bypass control*)
	HMI_227DSB : HMI_DI_Type; (*Doser Bypass control*)
	HMI_Beacon : HMI_Beacon_Type;
	HMI_BeaconHome : ARRAY[0..1] OF HMI_BeaconHome_Type; (*Reserved Home Page HMI V4.A.A.1.6.8*)
	HMI_GNS_LadderRestPosition : BOOL;
END_VAR
```

### HMI_ICO.var
```iecst
VAR
	HMI_ICO : HMI_ICO_Type;
END_VAR
```

### HMI_ITC.var
```iecst
(*INTERCHANGE PAGE*)
VAR
	HMI_ITC_PageDB : ARRAY[CST_MinITCPartner..CST_MaxITCPartner] OF HMI_ITC_Data_Type;
	HMI_ITC_Page : HMI_ITC_Page_Type;
	HMI_ITC_Partner_CFG : ARRAY[0..CST_MaxITCPartner] OF BOOL;
	HMI_MachineComm : HMI_MachineComm_Type;
END_VAR
```

### HMI_MAU.var
```iecst
VAR
	HMI_MAU_PB : ARRAY[MIN_PB_CFG..MAX_PB_CFG] OF PB_Type;
	HMI_MAU_SS2P : ARRAY[MIN_SS2P_CFG..MAX_SS2P_CFG] OF SS2P_Type;
END_VAR
(*GREASING/LUBRIFICATION*)
VAR
	HMI_201GPE : HMI_GreasingPump_Type;
	HMI_GrLb_PB : ARRAY[MIN_PB_CFG..MAX_PB_CFG] OF PB_Type;
	HMI_GrLb_Data : HMI_GrLb_Data_Type;
	HMI_GrLb_Data2 : HMI_GrLb_Data_Type; (*//V4.A.A.1.6.11*)
END_VAR
(*WHITE ROOM*)
VAR
	HMI_WhRoom_SS2P : ARRAY[MIN_SS2P_CFG..MAX_SS2P_CFG] OF SS2P_Type;
	HMI_FanBase : HMI_Fan_Type;
	HMI_FanFiller : HMI_Fan_Type;
	HMI_FanRinser : HMI_Fan_Type;
	HMI_FanTransfer : HMI_Fan_Type;
END_VAR
(*UPS*)
VAR
	HMI_UPS_ShutdownRequest : BOOL;
END_VAR
(*LIFT CONTAINERS*)
VAR
	HMI_205RVF : HMI_Analog_IN_Type;
	HMI_203RVF : HMI_Analog_IN_Type;
	HMI_205EVF : HMI_Valve_Type;
	HMI_LftCon_SS2P : ARRAY[MIN_SS2P_CFG..MAX_SS2P_CFG] OF SS2P_Type;
END_VAR
(*SAFE LOGIC*)
VAR
	HMI_SL_PB : HMI_SL_PB_Type;
	HMI_SL_Info : HMI_SL_Info_Type;
END_VAR
(*LUBRIFICATION*)
VAR
	HMI_MAU_ChlRns : HMI_MAU_ChlRns_Type; (*master nuovo*)
	HMI_LbCon_PB : ARRAY[MIN_PB_CFG..MAX_PB_CFG] OF PB_Type;
END_VAR
(*PLC*)
VAR
	HMI_TimeZoneOffset : INT;
	HMI_SDM_MachineStopped : BOOL; (*machine stopped 1.7.2b*)
	HMI_SDM_PLCAvailable : BOOL; (*information to HMI that SDM is active 1.7.2*)
	HMI_SDM_RequestInit : BOOL; (*SDM activation request,operator is in SDM page with machine stopped 1.7.2*)
	HMI_FSF : ARRAY[MIN_CFG_FSx..MAX_CFG_FSx] OF HMI_DI_Type;
END_VAR
(*TRAY DSEVICES*)
VAR
	HMI_209DSF : HMI_DI_Type; (*Tray Piston Inserted v1.4*)
	HMI_227CPB : HMI_Valve_Type; (*Tray Piston v1.4*)
END_VAR
(*EXHAUSTER //v1.7.4*)
VAR
	HMI_AFE : ARRAY[200..209] OF HMI_Motor_FC_Type; (*Filler aspirator //v1.7.5*)
	HMI_VFD_AFE : ARRAY[200..209] OF HMI_Danfoss_Diag_Type; (*Filler aspirator //v1.7.5*)
END_VAR
```

### HMI_MC.var
```iecst
VAR
	HMI_MC_MachineStatus : ST_HmiMachineStatus;
	HMI_AxisIndex : USINT; (*V4.A.A.1.7.0*)
	HMI_MC_GenericAxisDataNew : ARRAY[0..14] OF ST_HmiNewAxisData; (*vrma*)
	HMI_MC_GenericAxisData : ST_HmiAxisData;
	HMI_MC_AlarmList : ARRAY[0..9] OF STRING[50];
	HMI_MC_AxisPresent : ST_HmiAxisPresent;
	HMI_MC_EncoderDiagnostic : ST_HMIEncoderDiagnostic;
END_VAR
```

### HMI_MNM.var
```iecst
VAR
	HMI_MNM_PB : ARRAY[MIN_PB_CFG..MAX_PB_CFG] OF PB_Type;
	HMI_MNM_SS2P : ARRAY[MIN_SS2P_CFG..MAX_SS2P_CFG] OF SS2P_Type;
	HMI_MNM_MachineSpeedAct : REAL;
	HMI_MNM_MachineSpeedReq : REAL;
END_VAR
VAR CONSTANT
	HMI_MNM_MinMachineSpeed : REAL := 2000.0;
END_VAR
VAR
	HMI_MNM_MinMachineJogSpeed : REAL;
	HMI_MNM_MaxMachineJogSpeed : REAL;
	HMI_MNM_MinInMotionAdjustement : REAL;
	HMI_MNM_MaxInMotionAdjustement : REAL;
	HMI_MNM_MaxMachineSpeed : REAL;
	HMI_MNM_AxisPositionOffset : REAL;
	HMI_MNM_AxisStepByStepOffset : UINT;
	HMI_MNM_AxisInMotionAdjustment : REAL;
	HMI_MNM_MachinePosition : UINT;
	HMI_MNM_MachinePitch : REAL;
	HMI_MNM_AxisSelected : UINT;
	HMI_MNM_ConveyorSpeed : REAL;
	HMI_MNM_FlrSpeedWidget : HMI_SpeedWidget_Type;
	HMI_MNM_SmrSpeedWidget : HMI_SpeedWidget_Type;
	HMI_MNM_CamName : ARRAY[1..11] OF USINT; (*V4.A.A.1.7.0 v999hema*)
	HMI_MNM_MachineRunning : BOOL;
END_VAR
(*DMC*)
VAR
	HMI_MNM_NumOfDmcInTangentSector2 : USINT;
	HMI_MNM_NumOfDmcInTangentSector1 : USINT;
END_VAR
(*MOTORS*)
VAR
	HMI_InCvr : HMI_Motor_FC_Type; (*Infeed conveyor motor v1.7.4a*)
	HMI_OutCvr : HMI_Motor_FC_Type; (*Outfeed conveyor motor*)
END_VAR
(*DRIVERS*)
VAR
	HMI_VFD_InCvr : HMI_Danfoss_Diag_Type; (*Infeed conveyor VFD v1.7.4a*)
	HMI_VFD_OutCvr : HMI_Danfoss_Diag_Type; (*Outfeed conveyor VFD*)
END_VAR
(*DIGITAL INSTRUMENT*)
VAR
	HMI_241DSE : HMI_DI_Type; (*Caps Discharge*)
	HMI_230DSE : HMI_DI_Type; (*Spot safety*)
	HMI_236DSE : HMI_DI_Type; (*Outlet obstructed*)
	HMI_ContainerFallInlet1 : BOOL; (*Container fall at inlet 1*)
	HMI_ContainerFallInlet2 : BOOL; (*Container fall at inlet 2*)
	HMI_NoContainerInlet1 : BOOL; (*No container at Inlet 1*)
	HMI_NoContainerInlet2 : BOOL; (*No container at Inlet 2*)
	HMI_OutletFull : BOOL;
END_VAR
(*INLET SENSOR*)
VAR
	HMI_CloseInlet : HMI_DI_Type; (*v1.7.4a*)
	HMI_FarInlet : HMI_DI_Type; (*v1.7.4a*)
END_VAR
(*INLET CANS SENSOR*)
VAR
	HMI_InletSafetyLow1 : HMI_DI_Type;
	HMI_InletSafetyHigh1 : HMI_DI_Type;
	HMI_InletSafetyLow2 : HMI_DI_Type;
	HMI_InletSafetyHigh2 : HMI_DI_Type;
END_VAR
```

### HMI_MNT.var
```iecst
VAR
	HMI_MNT : HMI_MNT_Type;
END_VAR
```

### HMI_OPS.var
```iecst
VAR
	HMI_OPS_Zone : ARRAY[MIN_CFG_SafetyZone..MAX_CFG_SafetyZone] OF HMI_OPS_Zone_Type; (*1: Forward
2: Backward Inlet
3: Backward Outlet
4: Inlet Transfer Forward
5: Inlet Transfer Backward
6:
7: Filler Maintenance Inlet
8: Filler Maintenance Outlet/Capper Platform
9:
10:Transfer  Gate
11:Forward 2
12: Backward Inlet 2
13: Backward Outlet 2
14:
15:
16:Backward Rinser Inlet
17:Backward Rinser Outlet
18:Maintenance Rinser Outlet
19:
20:
21:Backward Pulp Doser
22:Backward Pulp Doser 2*)
	HMI_OPS_BufferZone : HMI_OPS_Zone_Type;
	HMI_OPS_GateDoor : ARRAY[0..1] OF HMI_GateDoor_Type; (*0: Inlet Gate
1: Outlet Gate*)
	HMI_OPS_Door : ARRAY[0..MAX_CFG_DoorConfiguration] OF HMI_OPS_Door_Type;
	HMI_OPS_DoorCabinet_Visibility : BOOL;
	HMI_OPS_DoorCabinet : ARRAY[1..5] OF HMI_OPS_Door_Type;
	HMI_OPS_Euchner : HMI_OPS_RfidAccess_Type;
	HMI_OPS_SafetySwitch : HMI_OPS_SafetySwitch_Type; (*V4.A.A.1.7.1*)
	HMI_OPS_BufferDoor : ARRAY[1..4] OF HMI_OPS_Door_Type; (*V4.A.A.1.6.12d*)
	HMI_OPS_Emergency : ARRAY[0..MAX_CFG_EmergencyConfiguration] OF HMI_OPS_Emergency_Type;
	HMI_OPS_Jog : ARRAY[0..MAX_CFG_JogConfiguration] OF HMI_OPS_Jog_Type;
	HMI_OPS_JogFwExt : HMI_OPS_Jog_Type; (*vrma106*)
	HMI_OPS_EmergencyBlower : HMI_OPS_Emergency_Type;
	HMI_OPS_EmergencyLabeller : HMI_OPS_Emergency_Type;
	HMI_OPS_EmergencyActis : HMI_OPS_Emergency_Type; (*V4.A.A.1.6.12*)
	HMI_OPS_EmergencyConveyor : HMI_OPS_Emergency_Type;
	HMI_OPS_EmergencyNitrodoser : HMI_OPS_Emergency_Type;
	HMI_OPS_EmergencyCrownFeeder : HMI_OPS_Emergency_Type;
	HMI_OPS_EmergencyCapsFeeder : HMI_OPS_Emergency_Type;
	HMI_OPS_ModeSelectorAdjustment : BOOL;
	HMI_OPS_ModeSelectorJog : BOOL; (*V4.A.A.1.6.13*)
	HMI_OPS_ModeSelectorAuto : BOOL; (*V4.A.A.1.6.13*)
	HMI_OPS_SafetyWidget : HMI_SafetyWidget_Type;
	HMI_207EVF : HMI_Valve_Type; (*Soffio Paratia automatica COP V4.A.A.1.6.12*)
	HMI_208CPF : HMI_Valve_Type; (*Paratia automatica COP V4.A.A.1.6.12*)
	HMI_208DSFX : HMI_DI_Type; (*Paratia automatica COP Aperta V4.A.A.1.6.12*)
	HMI_208DSFY : HMI_DI_Type; (*Paratia automatica COP Chiusa V4.A.A.1.6.12*)
	HMI_209DSFX : HMI_DI_Type; (*Paratia automatica COP Aperta V4.A.A.1.6.12*)
	HMI_209DSFY : HMI_DI_Type; (*Paratia automatica COP Chiusa V4.A.A.1.6.12*)
	HMI_209EVF : HMI_Valve_Type;
	HMI_OPS_Pictogram : HMI_OPS_Pictogram_Type;
	HMI_OPS_Cfg : CFG_OPS_Type;
	HMI_OPS_PB : ARRAY[MIN_PB_CFG..MAX_PB_CFG] OF PB_Type;
	HMI_OPS_SS2P : ARRAY[MIN_SS2P_CFG..MAX_SS2P_CFG] OF SS2P_Type; (*V4.A.A.1.6.12h*)
	HMI_OPS_ZoneComboString : STRING[250];
END_VAR
```

### HMI_RCP.var
```iecst
VAR RETAIN
	HMI_RCP_PRD_Mngt : RCP_Management_Type; (*Production recipe managment*)
END_VAR
```

### HMI_SFT.var
```iecst
VAR
	HMI_TotalBottleProduced : UDINT;
END_VAR
(*HMI Variables for Auto Step Acquisition*)
VAR
	HMI_StepAcquisition : StepAcquisition_Type;
END_VAR
(*VALVES*)
VAR
	HMI_StepAcquisition_BlowerLenght : StepAcquisition_Sensor_Type; (*v1.4*)
	HMI_SFT_SS3P : ARRAY[MIN_SS3P_CFG..MAX_SS3P_CFG] OF SS3P_Type;
	HMI_SFT_SS2P : ARRAY[MIN_SS2P_CFG..MAX_SS2P_CFG] OF SS2P_Type;
	HMI_SFT_PB : ARRAY[MIN_PB_CFG..MAX_PB_CFG] OF PB_Type;
	HMI_201CPB : HMI_Valve_Type;
	HMI_207CPF : HMI_Valve_Type; (*Roller Security Cam*)
	HMI_207CPB : HMI_Valve_Type; (*Nob Nos 1° Treatment*)
	HMI_215CPB : HMI_Valve_Type;
	HMI_210CPF : HMI_Valve_Type; (*v999hema*)
	HMI_202EVR : HMI_Valve_Type;
END_VAR
(*HMI Bottle Burst*)
VAR RETAIN
	HMI_SFT_BurstData : ARRAY[1..200] OF HMI_SFT_BurstData_Type;
END_VAR
(*HMI Variables For Container Check*)
VAR
	HMI_202DSF : HMI_Photocell_Type;
	HMI_203DSF : HMI_Photocell_Type;
	HMI_204DSF : HMI_Photocell_Type;
	HMI_207DSF : HMI_Photocell_Type;
	HMI_208DSF : HMI_Photocell_Type;
	HMI_204DSB : HMI_Photocell_Type; (*V4.A.A.1.6.11*)
END_VAR
(*HMI Variables for Dummy Container Piston Position Check*)
VAR
	HMI_ProductionSensorCheck1 : HMI_DI_Type;
	HMI_ProductionSensorCheck2 : HMI_DI_Type;
	HMI_SFT_NumberOfDmcInPosCheck : INT;
	HMI_SFT_NumberOfDummyInError : INT;
	HMI_ProductionSensorCheck3 : HMI_DI_Type;
END_VAR
(*COUNTERS*)
VAR RETAIN
	HMI_CounterDataPartial : CounterData_Type;
	HMI_CounterDataTotal : CounterData_Type;
END_VAR
VAR
	HMI_CounterCfgTotal : CounterCfg_Type;
	HMI_CounterCfgPartial : CounterCfg_Type;
END_VAR
```

### HMI_TNK.var
```iecst
VAR
	HMI_FMC_ActualFlowRate : REAL;
END_VAR
```

### HMI_B.var
```iecst
(*VALVES*)
VAR
	HMI_AVB : ARRAY[MIN_CFG_AVx..MAX_CFG_AVx] OF HMI_Valve_Type;
	HMI_RVB : ARRAY[MIN_CFG_RVx..MAX_CFG_RVx] OF HMI_Valve_Mod_Type;
	HMI_RMB : ARRAY[MIN_CFG_RMx..MAX_CFG_RMx] OF HMI_Valve_Mod_Type;
	HMI_HVB : ARRAY[MIN_CFG_HVx..MAX_CFG_HVx] OF HMI_Valve_Type; (*V4.A.A.1.6.12*)
	HMI_EVB : ARRAY[MIN_CFG_EVx..MAX_CFG_EVx] OF HMI_Valve_Type; (*v1.7.4*)
	HMI_206CPB : HMI_Valve_Type; (*Moovable Spray Control V4.A.A.1.7.0*)
	HMI_296CPB : HMI_Valve_Type; (*Moovable Cam ByPass Outlet Starwheel V4.A.A.1.7.0*)
	HMI_297CPB : HMI_Valve_Type; (*Moovable Cam ByPass Inlet Starwheel V4.A.A.1.7.0*)
	HMI_298CPB : HMI_Valve_Type; (*Moovable ByPass Starwheel Outlet Cam V4.A.A.1.7.0*)
	HMI_299CPB : HMI_Valve_Type; (*Moovable ByPass Starwheel Inlet Cam V4.A.A.1.7.0*)
	HMI_211CPB : HMI_Valve_Type; (*Doser ByPass Control RMH017*)
	HMI_212CPB : HMI_Valve_Type; (*Doser ByPass Control*)
	HMI_213CPB : HMI_Valve_Type; (*Doser ByPass Control*)
	HMI_219CPB : HMI_Valve_Type; (*Doser ByPass Control*)
END_VAR
(*INSTRUMENTS - DIGITAL*)
VAR
	HMI_PSB : ARRAY[MIN_CFG_PSx..MAX_CFG_PSx] OF HMI_DI_Type;
	HMI_LSB : ARRAY[MIN_CFG_LSx..MAX_CFG_LSx] OF HMI_DI_Type;
	HMI_HSB : ARRAY[MIN_CFG_HSx..MAX_CFG_HSx] OF HMI_DI_Type; (*V4.A.A.1.6.12*)
	HMI_FSB : ARRAY[MIN_CFG_FSx..MAX_CFG_FSx] OF HMI_DI_Type;
	HMI_QSB : ARRAY[MIN_CFG_QSx..MAX_CFG_QSx] OF HMI_DI_Type; (*v1.7.4*)
	HMI_202DSB : HMI_DI_Type; (*V4.A.A.1.7.0*)
	HMI_298DSB : HMI_DI_Type; (*V4.A.A.1.7.0*)
	HMI_299DSB : HMI_DI_Type; (*V4.A.A.1.7.0*)
	HMI_205DSB : HMI_DI_Type; (*V4.A.A.1.7.0*)
END_VAR
(*INSTRUMENTS - ANALOGIC*)
VAR
	HMI_CTB : ARRAY[MIN_CFG_CTx..MAX_CFG_CTx] OF HMI_Analog_IN_Mode_Type;
	HMI_QTB : ARRAY[MIN_CFG_QTx..MAX_CFG_QTx] OF HMI_Analog_IN_Type; (*v1.7.4*)
	HMI_FTB : ARRAY[MIN_CFG_FTx..MAX_CFG_FTx] OF HMI_Analog_IN_Type;
	HMI_TTB : ARRAY[MIN_CFG_TTx..MAX_CFG_TTx] OF HMI_Analog_IN_Type;
	HMI_PTB : ARRAY[MIN_CFG_PTx..MAX_CFG_PTx] OF HMI_Analog_IN_Type;
	HMI_LTB : ARRAY[MIN_CFG_LTx..MAX_CFG_LTx] OF HMI_Analog_IN_Type;
END_VAR
(*PIDs*)
VAR
	HMI_PID_PPB : ARRAY[MIN_CFG_PID_PPx..MAX_CFG_PID_PPx] OF HMI_PID_Type;
	HMI_PID_RVB : ARRAY[MIN_CFG_PID_RVx..MAX_CFG_PID_RVx] OF HMI_PID_Mode_Type;
	HMI_PID_RMB : ARRAY[MIN_CFG_PID_RMx..MAX_CFG_PID_RMx] OF HMI_PID_Mode_Type;
END_VAR
(*MOTORS*)
VAR
	HMI_MMB : ARRAY[MIN_CFG_VFD_MMx..MAX_CFG_VFD_MMx] OF HMI_Motor_FC_Type;
	HMI_VFD_MMB : ARRAY[MIN_CFG_VFD_MMx..MAX_CFG_VFD_MMx] OF HMI_Danfoss_Diag_Type;
	HMI_PPB : ARRAY[MIN_CFG_VFD_PPx..MAX_CFG_VFD_PPx] OF HMI_Motor_FC_Type;
	HMI_VFD_PPB : ARRAY[MIN_CFG_VFD_PPx..MAX_CFG_VFD_PPx] OF HMI_Danfoss_Diag_Type;
END_VAR
```

### HMI_C.var
```iecst
(*VALVES*)
VAR
	(*HMI_AVC : ARRAY[MIN_CFG_AVC..MAX_CFG_AVC] OF HMI_Valve_Type;*)
	HMI_RVC : ARRAY[MIN_CFG_RVx..MAX_CFG_RVx] OF HMI_Valve_Mod_Type;
	HMI_RMC : ARRAY[MIN_CFG_RMx..MAX_CFG_RMx] OF HMI_Valve_Mod_Type;
	HMI_HVC : ARRAY[MIN_CFG_HVx..MAX_CFG_HVx] OF HMI_Valve_Type; (*V4.A.A.1.6.12*)
END_VAR
(*INSTRUMENTS - DIGITAL*)
VAR
	HMI_PSC : ARRAY[MIN_CFG_PSx..MAX_CFG_PSx] OF HMI_DI_Type;
	HMI_LSC : ARRAY[MIN_CFG_LSx..MAX_CFG_LSx] OF HMI_DI_Type;
	HMI_HSC : ARRAY[MIN_CFG_HSx..MAX_CFG_HSx] OF HMI_DI_Type; (*V4.A.A.1.6.12*)
	HMI_FSC : ARRAY[MIN_CFG_FSx..MAX_CFG_FSx] OF HMI_DI_Type;
END_VAR
(*INSTRUMENTS - ANALOGIC*)
VAR
	HMI_CTC : ARRAY[MIN_CFG_CTx..MAX_CFG_CTx] OF HMI_Analog_IN_Mode_Type;
	HMI_QTC : ARRAY[MIN_CFG_QTx..MAX_CFG_QTx] OF HMI_Analog_IN_Type;
	HMI_FTC : ARRAY[MIN_CFG_FTx..MAX_CFG_FTx] OF HMI_Analog_IN_Type;
	HMI_TTC : ARRAY[MIN_CFG_TTx..MAX_CFG_TTx] OF HMI_Analog_IN_Type;
	HMI_PTC : ARRAY[MIN_CFG_PTx..MAX_CFG_PTx] OF HMI_Analog_IN_Type;
	HMI_LTC : ARRAY[MIN_CFG_LTx..MAX_CFG_LTx] OF HMI_Analog_IN_Type;
END_VAR
(*PIDs*)
VAR
	HMI_PID_PPC : ARRAY[MIN_CFG_PID_PPx..MAX_CFG_PID_PPx] OF HMI_PID_Mode_Type;
	HMI_PID_RVC : ARRAY[MIN_CFG_PID_RVx..MAX_CFG_PID_RVx] OF HMI_PID_Mode_Type;
	HMI_PID_RMC : ARRAY[MIN_CFG_PID_RMx..MAX_CFG_PID_RMx] OF HMI_PID_Mode_Type;
END_VAR
(*MOTORS*)
VAR
	HMI_MMC : ARRAY[MIN_CFG_VFD_MMx..MAX_CFG_VFD_MMx] OF HMI_Motor_FC_Type;
	HMI_VFD_MMC : ARRAY[MIN_CFG_VFD_MMx..MAX_CFG_VFD_MMx] OF HMI_Danfoss_Diag_Type;
	HMI_PPC : ARRAY[MIN_CFG_VFD_PPx..MAX_CFG_VFD_PPx] OF HMI_Motor_FC_Type;
	HMI_VFD_PPC : ARRAY[MIN_CFG_VFD_PPx..MAX_CFG_VFD_PPx] OF HMI_Danfoss_Diag_Type;
END_VAR
```

### HMI_E.var
```iecst
(*VALVES*)
VAR
	HMI_AVE : ARRAY[MIN_CFG_AVx..MAX_CFG_AVx] OF HMI_Valve_Type;
	HMI_HVE : ARRAY[MIN_CFG_HVx..MAX_CFG_HVx] OF HMI_Valve_Type; (*V4.A.A.1.6.12*)
	HMI_RVE : ARRAY[MIN_CFG_RVx..MAX_CFG_RVx] OF HMI_Valve_Mod_Type;
	HMI_RME : ARRAY[MIN_CFG_RMx..MAX_CFG_RMx] OF HMI_Valve_Mod_Type;
END_VAR
(*INSTRUMENTS - DIGITAL*)
VAR
	HMI_PSE : ARRAY[MIN_CFG_PSx..MAX_CFG_PSx] OF HMI_DI_Type;
	HMI_LSE : ARRAY[MIN_CFG_LSx..MAX_CFG_LSx] OF HMI_DI_Type;
	HMI_FSE : ARRAY[MIN_CFG_FSx..MAX_CFG_FSx] OF HMI_DI_Type;
	HMI_HSE : ARRAY[MIN_CFG_HSx..MAX_CFG_HSx] OF HMI_DI_Type; (*V4.A.A.1.6.12*)
END_VAR
(*INSTRUMENTS - ANALOGIC*)
VAR
	HMI_CTE : ARRAY[MIN_CFG_CTx..MAX_CFG_CTx] OF HMI_Analog_Multiscale_Type;
	HMI_QTE : ARRAY[MIN_CFG_QTx..MAX_CFG_QTx] OF HMI_Analog_IN_Type;
	HMI_FTE : ARRAY[MIN_CFG_FTx..MAX_CFG_FTx] OF HMI_Analog_IN_Type;
	HMI_TTE : ARRAY[MIN_CFG_TTx..MAX_CFG_TTx] OF HMI_Analog_IN_Type;
	HMI_PTE : ARRAY[MIN_CFG_PTx..MAX_CFG_PTx] OF HMI_Analog_IN_Type;
	HMI_LTE : ARRAY[MIN_CFG_LTx..MAX_CFG_LTx] OF HMI_Analog_IN_Type;
	HMI_204PTE : HMI_Analog_IN_Type;
	HMI_205PTE : HMI_Analog_IN_Type;
	HMI_206PTE : HMI_Analog_IN_Type;
	HMI_207PTE : HMI_Analog_IN_Type; (*V4.A.A.1.7.6*)
END_VAR
(*PIDs*)
VAR
	HMI_PID_PPE : ARRAY[MIN_CFG_PID_PPx..MAX_CFG_PID_PPx] OF HMI_PID_Mode_Type;
	HMI_PID_RVE : ARRAY[MIN_CFG_PID_RVx..MAX_CFG_PID_RVx] OF HMI_PID_Mode_Type;
	HMI_PID_RME : ARRAY[MIN_CFG_PID_RMx..MAX_CFG_PID_RMx] OF HMI_PID_Mode_Type;
END_VAR
(*MOTORS*)
VAR
	HMI_MME : ARRAY[MIN_CFG_VFD_MMx..MAX_CFG_VFD_MMx] OF HMI_Motor_FC_Type;
	HMI_VFD_MME : ARRAY[MIN_CFG_VFD_MMx..MAX_CFG_VFD_MMx] OF HMI_Danfoss_Diag_Type;
	HMI_VFD_PPE : ARRAY[MIN_CFG_VFD_PPx..MAX_CFG_VFD_PPx] OF HMI_Danfoss_Diag_Type;
	HMI_PPE : ARRAY[MIN_CFG_VFD_PPx..MAX_CFG_VFD_PPx] OF HMI_Motor_FC_Type;
END_VAR
(*HEATERS*)
VAR
	HMI_EHE : ARRAY[MIN_CFG_AVx..MAX_CFG_AVx] OF HMI_Motor_Type;
END_VAR
```

### HMI_S.var
```iecst
(*VALVES*)
VAR
	HMI_AVS : ARRAY[MIN_CFG_AVx..MAX_CFG_AVx] OF HMI_Valve_Type;
	HMI_RVS : ARRAY[MIN_CFG_RVx..MAX_CFG_RVx] OF HMI_Valve_Mod_Type;
	HMI_RMS : ARRAY[MIN_CFG_RMx..MAX_CFG_RMx] OF HMI_Valve_Mod_Type;
END_VAR
(*INSTRUMENTS - DIGITAL*)
VAR
	HMI_PSS : ARRAY[MIN_CFG_PSx..MAX_CFG_PSx] OF HMI_DI_Type;
	HMI_LSS : ARRAY[MIN_CFG_LSx..MAX_CFG_LSx] OF HMI_DI_Type;
	HMI_FSS : ARRAY[MIN_CFG_FSx..MAX_CFG_FSx] OF HMI_DI_Type;
END_VAR
(*INSTRUMENTS - ANALOGIC*)
VAR
	HMI_CTS : ARRAY[MIN_CFG_CTx..MAX_CFG_CTx] OF HMI_Analog_IN_Mode_Type;
	HMI_QTS : ARRAY[MIN_CFG_QTx..MAX_CFG_QTx] OF HMI_Analog_IN_Type;
	HMI_FTS : ARRAY[MIN_CFG_FTx..MAX_CFG_FTx] OF HMI_Analog_IN_Type;
	HMI_TTS : ARRAY[MIN_CFG_TTx..MAX_CFG_TTx] OF HMI_Analog_IN_Type;
	HMI_PTS : ARRAY[MIN_CFG_PTx..MAX_CFG_PTx] OF HMI_Analog_IN_Type;
	HMI_LTS : ARRAY[MIN_CFG_LTx..MAX_CFG_LTx] OF HMI_Analog_IN_Type;
END_VAR
(*PIDs*)
VAR
	HMI_PID_PPS : ARRAY[MIN_CFG_PID_PPx..MAX_CFG_PID_PPx] OF HMI_PID_Mode_Type;
	HMI_PID_RVS : ARRAY[MIN_CFG_PID_RVx..MAX_CFG_PID_RVx] OF HMI_PID_Mode_Type;
	HMI_PID_RMS : ARRAY[MIN_CFG_PID_RMx..MAX_CFG_PID_RMx] OF HMI_PID_Mode_Type;
END_VAR
(*MOTORS*)
VAR
	HMI_VFD_MMS : ARRAY[MIN_CFG_VFD_MMx..MAX_CFG_VFD_MMx] OF HMI_Danfoss_Diag_Type;
	HMI_VFD_PPS : ARRAY[MIN_CFG_VFD_PPx..MAX_CFG_VFD_PPx] OF HMI_Danfoss_Diag_Type;
	HMI_PPS : ARRAY[MIN_CFG_VFD_PPx..MAX_CFG_VFD_PPx] OF HMI_Motor_FC_Type;
END_VAR
(*HEATERS*)
VAR
	HMI_EHS : ARRAY[MIN_CFG_AVx..MAX_CFG_AVx] OF HMI_Motor_Type;
END_VAR
```

### HMI_X.var
```iecst
(*VALVES*)
VAR
	HMI_AVX : ARRAY[MIN_CFG_AVx..MAX_CFG_AVx] OF HMI_Valve_Type;
	HMI_RVX : ARRAY[MIN_CFG_RVx..MAX_CFG_RVx] OF HMI_Valve_Mod_Type;
	HMI_RMX : ARRAY[MIN_CFG_RMx..MAX_CFG_RMx] OF HMI_Valve_Mod_Type;
END_VAR
(*INSTRUMENTS - DIGITAL*)
VAR
	HMI_PSX : ARRAY[MIN_CFG_PSx..MAX_CFG_PSx] OF HMI_DI_Type;
	HMI_LSX : ARRAY[MIN_CFG_LSx..MAX_CFG_LSx] OF HMI_DI_Type;
	HMI_FSX : ARRAY[MIN_CFG_FSx..MAX_CFG_FSx] OF HMI_DI_Type;
	HMI_TSX : ARRAY[MIN_CFG_FSx..MAX_CFG_FSx] OF HMI_DI_Type; (*//V4.A.A.1.7.4*)
END_VAR
(*INSTRUMENTS - ANALOGIC*)
VAR
	HMI_CTX : ARRAY[MIN_CFG_CTx..MAX_CFG_CTx] OF HMI_Analog_IN_Mode_Type;
	HMI_QTX : ARRAY[MIN_CFG_QTx..MAX_CFG_QTx] OF HMI_Analog_IN_Type;
	HMI_FTX : ARRAY[MIN_CFG_FTx..MAX_CFG_FTx] OF HMI_Analog_IN_Type;
	HMI_TTX : ARRAY[MIN_CFG_TTx..MAX_CFG_TTx] OF HMI_Analog_IN_Type;
	HMI_PTX : ARRAY[MIN_CFG_PTx..MAX_CFG_PTx] OF HMI_Analog_IN_Type;
	HMI_LTX : ARRAY[MIN_CFG_LTx..MAX_CFG_LTx] OF HMI_Analog_IN_Type;
END_VAR
(*PIDs*)
VAR
	HMI_PID_PPX : ARRAY[MIN_CFG_PID_PPx..MAX_CFG_PID_PPx] OF HMI_PID_Mode_Type;
	HMI_PID_RVX : ARRAY[MIN_CFG_PID_RVx..MAX_CFG_PID_RVx] OF HMI_PID_Mode_Type;
	HMI_PID_RMX : ARRAY[MIN_CFG_PID_RMx..MAX_CFG_PID_RMx] OF HMI_PID_Mode_Type;
END_VAR
(*MOTORS*)
VAR
	HMI_MMX : ARRAY[MIN_CFG_VFD_MMx..MAX_CFG_VFD_MMx] OF HMI_Motor_FC_Type;
	HMI_VFD_MMX : ARRAY[MIN_CFG_VFD_MMx..MAX_CFG_VFD_MMx] OF HMI_Danfoss_Diag_Type;
	HMI_PPX : ARRAY[MIN_CFG_VFD_PPx..MAX_CFG_VFD_PPx] OF HMI_Motor_FC_Type;
	HMI_VFD_PPX : ARRAY[MIN_CFG_VFD_PPx..MAX_CFG_VFD_PPx] OF HMI_Danfoss_Diag_Type;
END_VAR
```

### HMI.var
```iecst
VAR RETAIN
	HMI_OPT_SS2P : ARRAY[MIN_SS2P_CFG..MAX_SS2P_CFG] OF SS2P_Type;
END_VAR
VAR
	HMI_MachineId : STRING[12];
	HMI_MachinePlcVersion : STRING[15]; (*V4.A.A.1.6.13*)
	HMI_MachineSafetyVersion : STRING[15]; (*V4.A.A.1.6.13*)
	HMI_ScreenTouched : BOOL;
	HMI_ApcoPresent : BOOL;
	HMI_214DSF : HMI_DI_Type; (*Head 1 Pulp Doser sensor  //v999hema*)
	HMI_IcoPresent : BOOL;
	HMI_CounterHome : HMI_CounterHome_Type; (*V4.A.A.1.6.8*)
END_VAR
```

### HMI_BTC.var - not listed in the package file held
```iecst
(*BOTTLE BOTTOM COOLING*)
VAR
	HMI_BTC_PB : ARRAY[MIN_PB_CFG..MAX_PB_CFG] OF PB_Type;
	HMI_BTC_SS2P : ARRAY[MIN_SS2P_CFG..MAX_SS2P_CFG] OF SS2P_Type;
	HMI_BTC_SS3P : ARRAY[MIN_SS3P_CFG..MAX_SS3P_CFG] OF SS3P_Type;
	HMI_BTC_State : HMI_BTC_State_Type;
	HMI_BTC_UVL : ARRAY[200..201] OF HMI_Motor_Type;
END_VAR
```

### Package Logical/02_HMI/0210_PAR - Parameters

### Program Logical/02_HMI/0210_PAR/PAR (IEC) - PAR Main Program - C#6 - 200ms

#### PAR.st - Init, cyclic code
```iecst
PROGRAM _INIT
//Call all the option parameters
	HMI_PAO_2;

	//Call all the parameters structure for HMI (RCP excluded)
	HMI_PAC_1;
	HMI_PAM_1;
	HMI_PAM_3;
	HMI_PAM_A1;
	HMI_PAM_B1;
	HMI_PAM_C1;
	HMI_PAM_D1;
	HMI_PAT_1;

	//Call all the parameters configuration structure for HMI (RCP excluded)
	HMI_CFG_PAC_1;
	HMI_CFG_PAM_1;
	HMI_CFG_PAM_3;
	HMI_CFG_PAM_A1;
	HMI_CFG_PAM_B1;
	HMI_CFG_PAM_C1;
	HMI_CFG_PAM_D1;
	HMI_CFG_PAT_1;
END_PROGRAM

PROGRAM _CYCLIC
	HMI_PB[PB_PAR_Initialization].Visibility	:= TRUE;
	HMI_PB[PB_PAR_Initialization].Enable		:= TRUE;

	IF VAR_PAR_Initialization THEN
		HMI_PAC_1_Init;
		HMI_PAM_1_Init;
		HMI_PAM_3_Init;
		HMI_PAM_A1_Init;
		HMI_PAM_B1_Init;
		HMI_PAM_C1_Init;
		HMI_PAM_D1_Init;
		HMI_PAT_1_Init;
		VAR_PAR_Initialization	:= FALSE;
	END_IF

	TMR_TON_ParInitialization(IN	:= HMI_PB[PB_PAR_Initialization].ON,
								PT := t#5s);

	IF CFG_Par.Process.BlendFill THEN
		FlrCrb.HMI_ParInitialization	:= HMI_PB[PB_PAR_Initialization].ON;
	ELSIF CFG_Par.Process.InternalSkid THEN
		FlrSkd.HMI_ParInitialization	:= HMI_PB[PB_PAR_Initialization].ON;
	END_IF

	IF TMR_TON_ParInitialization.Q THEN
		VAR_PAR_Initialization			:= TRUE;
	END_IF

	HMI_PB[PB_PAR_Initialization].Blink		:= HMI_PB[PB_PAR_Initialization].ON AND NOT TMR_TON_ParInitialization.Q;
	HMI_PB[PB_PAR_Initialization].LampON	:= VAR_PAR_Initialization OR TMR_TON_ParInitialization.Q;
END_PROGRAM
```

#### HMI_PAC_1.st
```iecst
(*HMI_PAC_1 Initialization Action for Filler PLC*)
(*Author = UTERF*)
(*DB Version : 0.11*)
(*File Version : 3,17*)

ACTION HMI_PAC_1_Init :
        HMI_PAC_1._000 := 0;
        HMI_PAC_1._001 := 20;
        HMI_PAC_1._002 := 200;
        HMI_PAC_1._003 := 0;
        HMI_PAC_1._004 := 1;
        HMI_PAC_1._005 := 1;
        HMI_PAC_1._006 := 1;
        HMI_PAC_1._007 := 210;
        HMI_PAC_1._008 := 105;
        HMI_PAC_1._009 := 0;
        HMI_PAC_1._013 := 205;
        HMI_PAC_1._014 := 0;
        HMI_PAC_1._015 := 0;
        HMI_PAC_1._016 := 0;
        HMI_PAC_1._017 := 0;
        HMI_PAC_1._018 := 0;
        HMI_PAC_1._019 := 89;
        HMI_PAC_1._020 := 118;
        HMI_PAC_1._021 := 0;
        HMI_PAC_1._022 := 0;
        HMI_PAC_1._023 := 0;
        HMI_PAC_1._024 := 0;
        HMI_PAC_1._025 := 0;
        HMI_PAC_1._045 := 0;
        HMI_PAC_1._070 := 0;
        HMI_PAC_1._071 := 0;
        HMI_PAC_1._100 := 91;
        HMI_PAC_1._101 := 75;
        HMI_PAC_1._102 := 5;
        HMI_PAC_1._103 := 0;
        HMI_PAC_1._104 := 85;
        HMI_PAC_1._105 := 0;
        HMI_PAC_1._106 := 0;
        HMI_PAC_1._107 := 0;
        HMI_PAC_1._108 := 0;
        HMI_PAC_1._110 := 0;
        HMI_PAC_1._111 := 0;
        HMI_PAC_1._112 := 0;
        HMI_PAC_1._113 := 0;
        HMI_PAC_1._114 := 0;
        HMI_PAC_1._115 := 0;
        HMI_PAC_1._117 := 0;
        HMI_PAC_1._118 := 0;
        HMI_PAC_1._120 := 0;
        HMI_PAC_1._121 := 0;
        HMI_PAC_1._122 := 0;
        HMI_PAC_1._123 := 0;
        HMI_PAC_1._124 := 0;
        HMI_PAC_1._125 := 0;
        HMI_PAC_1._126 := 0;
        HMI_PAC_1._127 := 0;
        HMI_PAC_1._128 := 0;
        HMI_PAC_1._129 := 1;
        HMI_PAC_1._130 := 33;
        HMI_PAC_1._131 := 1;
        HMI_PAC_1._132 := 0;
        HMI_PAC_1._133 := 1;
        HMI_PAC_1._134 := 1;
        HMI_PAC_1._145 := 0;
        HMI_PAC_1._146 := 0;
        HMI_PAC_1._150 := 6;
        HMI_PAC_1._151 := 1;
        HMI_PAC_1._152 := 74;
        HMI_PAC_1._200 := 0;
        HMI_PAC_1._201 := 0;
        HMI_PAC_1._202 := 0;
        HMI_PAC_1._203 := 0;
        HMI_PAC_1._204 := 0;
        HMI_PAC_1._205 := 0;
        HMI_PAC_1._206 := 0;
        HMI_PAC_1._207 := 0;
        HMI_PAC_1._208 := 0;
        HMI_PAC_1._209 := 0;
        HMI_PAC_1._210 := 0;
        HMI_PAC_1._211 := 0;
        HMI_PAC_1._212 := 0;
        HMI_PAC_1._213 := 0;
        HMI_PAC_1._214 := 0;
        HMI_PAC_1._215 := 0;
        HMI_PAC_1._219 := 0;
        HMI_PAC_1._220 := 0;
        HMI_PAC_1._245 := 0;
        HMI_PAC_1._246 := 0;
        HMI_PAC_1._300 := 0;
        HMI_PAC_1._301 := 0;
        HMI_PAC_1._302 := 0;
        HMI_PAC_1._303 := 0;
        HMI_PAC_1._304 := 0;
        HMI_PAC_1._305 := 0;
        HMI_PAC_1._306 := 0;
        HMI_PAC_1._307 := 0;
        HMI_PAC_1._400 := 0;
        HMI_PAC_1._401 := 0;
        HMI_PAC_1._402 := 0;
        HMI_PAC_1._403 := 0;
        HMI_PAC_1._404 := 0;
        HMI_PAC_1._405 := 0;
        HMI_PAC_1._406 := 0;
        HMI_PAC_1._407 := 0;
        HMI_PAC_1._408 := 0;
        HMI_PAC_1._409 := 0;
        HMI_PAC_1._410 := 0;
        HMI_PAC_1._411 := 0;
        HMI_PAC_1._412 := 0;
        HMI_PAC_1._413 := 0;
        HMI_PAC_1._415 := 0;
        HMI_PAC_1._416 := 0;
        HMI_PAC_1._417 := 0;
        HMI_PAC_1._418 := 0;
        HMI_PAC_1._419 := 0;
        HMI_PAC_1._420 := 0;
        HMI_PAC_1._422 := 0;
        HMI_PAC_1._423 := 0;
        HMI_PAC_1._500 := 0;
        HMI_PAC_1._501 := 0;
        HMI_PAC_1._502 := 0;
        HMI_PAC_1._503 := 0;
        HMI_PAC_1._504 := 0;
        HMI_PAC_1._505 := 0;
        HMI_PAC_1._510 := 0;
        HMI_PAC_1._600 := 0;
        HMI_PAC_1._601 := 0;
        HMI_PAC_1._605 := 0;
        HMI_PAC_1._606 := 0;
        HMI_PAC_1._610 := 0;
        HMI_PAC_1._620 := 0;
        HMI_PAC_1._621 := 0;
        HMI_PAC_1._622 := 0;
        HMI_PAC_1._623 := 0;
        HMI_PAC_1._700 := 0;
        HMI_PAC_1._701 := 0;
        HMI_PAC_1._702 := 0;
        HMI_PAC_1._703 := 0;
        HMI_PAC_1._704 := 1;
        HMI_PAC_1._705 := 1;
        HMI_PAC_1._706 := 1;
        HMI_PAC_1._800 := 0;
END_ACTION
```

#### HMI_PAM_1.st
```iecst
(*HMI_PAM_1 Initialization Action for Filler PLC*)
(*Author = ????*)
(*DB Version : 0.10*)
(*File Version : 3.29*)

ACTION HMI_PAM_1_Init :
        HMI_PAM_1._000 := 50;
        HMI_PAM_1._001 := 20000;
        HMI_PAM_1._002 := 60;
        HMI_PAM_1._003 := 5000;
        HMI_PAM_1._004 := 8000;
        HMI_PAM_1._005 := 5000;
        HMI_PAM_1._006 := 25000;
        HMI_PAM_1._007 := 15000;
        HMI_PAM_1._008 := 20000;
        HMI_PAM_1._009 := 20000;
        HMI_PAM_1._010 := 1500;
        HMI_PAM_1._011 := 8;
        HMI_PAM_1._012 := 8;
        HMI_PAM_1._013 := 0.13;
        HMI_PAM_1._014 := 20000;
        HMI_PAM_1._015 := 20000;
        HMI_PAM_1._020 := 55200;
        HMI_PAM_1._021 := 400;
        HMI_PAM_1._022 := 2;
        HMI_PAM_1._023 := 600;
        HMI_PAM_1._030 := 300;
        HMI_PAM_1._031 := 2;
        HMI_PAM_1._032 := 2;
        HMI_PAM_1._036 := 0;
        HMI_PAM_1._040 := 300;
        HMI_PAM_1._041 := 5;
        HMI_PAM_1._044 := 0;
        HMI_PAM_1._045 := 0;
        HMI_PAM_1._046 := 0;
        HMI_PAM_1._047 := 0;
        HMI_PAM_1._048 := 10;
        HMI_PAM_1._049 := 1;
        HMI_PAM_1._050 := 60;
        HMI_PAM_1._051 := 0;
        HMI_PAM_1._052 := 0;
        HMI_PAM_1._053 := 0;
        HMI_PAM_1._054 := 0;
        HMI_PAM_1._055 := 10000;
        HMI_PAM_1._056 := 20000;
        HMI_PAM_1._057 := 0;
        HMI_PAM_1._058 := 0;
        HMI_PAM_1._060 := 5;
        HMI_PAM_1._061 := 100;
        HMI_PAM_1._065 := 50;
        HMI_PAM_1._080 := 0;
        HMI_PAM_1._081 := 0;
        HMI_PAM_1._082 := 0;
        HMI_PAM_1._083 := 0;
        HMI_PAM_1._084 := 0;
        HMI_PAM_1._085 := 0;
        HMI_PAM_1._086 := 3;
        HMI_PAM_1._087 := 3;
        HMI_PAM_1._088 := 3;
        HMI_PAM_1._089 := 3;
        HMI_PAM_1._090 := 1000000;
        HMI_PAM_1._091 := 40000;
        HMI_PAM_1._092 := 3.2;
        HMI_PAM_1._093 := 3.2;
        HMI_PAM_1._100 := 0;
        HMI_PAM_1._101 := 0;
        HMI_PAM_1._102 := 0;
        HMI_PAM_1._103 := 100;
        HMI_PAM_1._104 := 100;
        HMI_PAM_1._105 := 2;
        HMI_PAM_1._106 := 15;
        HMI_PAM_1._107 := 10;
        HMI_PAM_1._108 := 5;
        HMI_PAM_1._109 := 5;
        HMI_PAM_1._110 := 25;
        HMI_PAM_1._111 := 15;
        HMI_PAM_1._112 := 30;
        HMI_PAM_1._113 := 20;
        HMI_PAM_1._114 := 2;
        HMI_PAM_1._115 := 30;
        HMI_PAM_1._116 := 10;
        HMI_PAM_1._117 := 20;
        HMI_PAM_1._118 := 30;
        HMI_PAM_1._119 := 0;
        HMI_PAM_1._120 := 0;
        HMI_PAM_1._130 := 0;
        HMI_PAM_1._131 := 0;
        HMI_PAM_1._140 := 0;
        HMI_PAM_1._141 := 0;
        HMI_PAM_1._142 := 0;
        HMI_PAM_1._143 := 0;
        HMI_PAM_1._144 := 0;
        HMI_PAM_1._150 := 0;
        HMI_PAM_1._151 := 0;
        HMI_PAM_1._152 := 0;
        HMI_PAM_1._153 := 0;
        HMI_PAM_1._154 := 0;
        HMI_PAM_1._155 := 0;
        HMI_PAM_1._156 := 0;
        HMI_PAM_1._160 := 0;
        HMI_PAM_1._161 := 0;
        HMI_PAM_1._162 := 0;
        HMI_PAM_1._163 := 0;
        HMI_PAM_1._164 := 0;
        HMI_PAM_1._165 := 0;
        HMI_PAM_1._166 := 0;
        HMI_PAM_1._170 := 0;
        HMI_PAM_1._171 := 0;
        HMI_PAM_1._172 := 0;
        HMI_PAM_1._173 := 0;
        HMI_PAM_1._174 := 0;
        HMI_PAM_1._175 := 0;
        HMI_PAM_1._180 := 0;
        HMI_PAM_1._181 := 0;
        HMI_PAM_1._200 := 0;
        HMI_PAM_1._201 := 0;
        HMI_PAM_1._202 := 0;
        HMI_PAM_1._203 := 0;
        HMI_PAM_1._204 := 0;
        HMI_PAM_1._215 := 200;
        HMI_PAM_1._216 := 100;
        HMI_PAM_1._217 := 0;
        HMI_PAM_1._218 := 0;
        HMI_PAM_1._220 := 0;
        HMI_PAM_1._221 := 0;
        HMI_PAM_1._222 := 0;
        HMI_PAM_1._223 := 0;
        HMI_PAM_1._224 := 0;
        HMI_PAM_1._235 := 100;
        HMI_PAM_1._236 := 50;
        HMI_PAM_1._237 := 0;
        HMI_PAM_1._238 := 0;
        HMI_PAM_1._250 := 115;
        HMI_PAM_1._251 := 115;
        HMI_PAM_1._260 := 0;
        HMI_PAM_1._261 := 0;
        HMI_PAM_1._262 := 0;
        HMI_PAM_1._263 := 0;
        HMI_PAM_1._264 := 0;
        HMI_PAM_1._265 := 0;
        HMI_PAM_1._266 := 1;
        HMI_PAM_1._267 := 0;
        HMI_PAM_1._268 := 0;
        HMI_PAM_1._269 := 2.42;
        HMI_PAM_1._270 := 2.42;
        HMI_PAM_1._271 := 2.42;
        HMI_PAM_1._272 := 50;
        HMI_PAM_1._273 := 50;
        HMI_PAM_1._274 := 50;
        HMI_PAM_1._275 := 20;
        HMI_PAM_1._276 := 20;
        HMI_PAM_1._277 := 20;
        HMI_PAM_1._300 := 50;
        HMI_PAM_1._301 := 60;
        HMI_PAM_1._302 := 80;
        HMI_PAM_1._305 := 50;
        HMI_PAM_1._306 := 60;
        HMI_PAM_1._307 := 80;
        HMI_PAM_1._310 := 50;
        HMI_PAM_1._311 := 60;
        HMI_PAM_1._312 := 80;
        HMI_PAM_1._315 := 60;
        HMI_PAM_1._316 := 65;
        HMI_PAM_1._317 := 80;
        HMI_PAM_1._320 := 50;
        HMI_PAM_1._321 := 60;
        HMI_PAM_1._322 := 80;
        HMI_PAM_1._396 := 0;
        HMI_PAM_1._397 := 0;
        HMI_PAM_1._398 := 0;
        HMI_PAM_1._399 := 0;
        HMI_PAM_1._400 := 220;
        HMI_PAM_1._401 := 40;
        HMI_PAM_1._402 := 10;
        HMI_PAM_1._403 := 1;
        HMI_PAM_1._404 := 96;
        HMI_PAM_1._405 := 276;
        HMI_PAM_1._406 := 0;
        HMI_PAM_1._407 := 1;
        HMI_PAM_1._408 := 0;
        HMI_PAM_1._409 := 0;
        HMI_PAM_1._410 := 0;
        HMI_PAM_1._411 := 0;
        HMI_PAM_1._412 := 0;
        HMI_PAM_1._413 := 0;
        HMI_PAM_1._414 := 0;
        HMI_PAM_1._415 := 0;
        HMI_PAM_1._416 := 0;
        HMI_PAM_1._417 := 0;
        HMI_PAM_1._418 := 0;
        HMI_PAM_1._419 := 0;
        HMI_PAM_1._420 := 0;
        HMI_PAM_1._421 := 0;
        HMI_PAM_1._422 := 0;
        HMI_PAM_1._423 := 0;
        HMI_PAM_1._424 := 0;
        HMI_PAM_1._425 := 0;
        HMI_PAM_1._426 := 0;
        HMI_PAM_1._427 := 0;
        HMI_PAM_1._428 := 0;
        HMI_PAM_1._429 := 0;
        HMI_PAM_1._430 := 0;
        HMI_PAM_1._431 := 0;
        HMI_PAM_1._432 := 0;
        HMI_PAM_1._433 := 0;
        HMI_PAM_1._434 := 0;
        HMI_PAM_1._435 := 0;
        HMI_PAM_1._436 := 0;
        HMI_PAM_1._437 := 0;
        HMI_PAM_1._438 := 0;
        HMI_PAM_1._439 := 0;
        HMI_PAM_1._450 := 0;
        HMI_PAM_1._451 := 0;
        HMI_PAM_1._452 := 0;
        HMI_PAM_1._453 := 0;
        HMI_PAM_1._454 := 0;
        HMI_PAM_1._500 := 5;
        HMI_PAM_1._501 := 5;
        HMI_PAM_1._502 := 5;
        HMI_PAM_1._503 := 5;
        HMI_PAM_1._504 := 5;
        HMI_PAM_1._505 := 5;
        HMI_PAM_1._506 := 5;
        HMI_PAM_1._507 := 5;
        HMI_PAM_1._508 := 5;
        HMI_PAM_1._509 := 5;
        HMI_PAM_1._510 := 5;
        HMI_PAM_1._511 := 5;
        HMI_PAM_1._512 := 5;
        HMI_PAM_1._513 := 5;
        HMI_PAM_1._514 := 5;
        HMI_PAM_1._515 := 5;
        HMI_PAM_1._516 := 5;
        HMI_PAM_1._517 := 5;
        HMI_PAM_1._518 := 5;
        HMI_PAM_1._519 := 5;
        HMI_PAM_1._520 := 5;
        HMI_PAM_1._521 := 5;
        HMI_PAM_1._524 := 5;
        HMI_PAM_1._525 := 5;
        HMI_PAM_1._526 := 5;
        HMI_PAM_1._527 := 5;
        HMI_PAM_1._550 := 30;
        HMI_PAM_1._551 := 10;
        HMI_PAM_1._559 := 0;
        HMI_PAM_1._560 := 1;
        HMI_PAM_1._561 := 0;
        HMI_PAM_1._562 := 1;
        HMI_PAM_1._563 := 3;
        HMI_PAM_1._564 := 0;
        HMI_PAM_1._565 := 0;
        HMI_PAM_1._566 := 0;
        HMI_PAM_1._567 := 0;
        HMI_PAM_1._568 := 0;
        HMI_PAM_1._569 := 0;
        HMI_PAM_1._900 := 0;
END_ACTION
```

#### HMI_PAM_3.st
```iecst
(*HMI_PAM_3 Initialization Action for Filler PLC*)
(*Author = ????*)
(*DB Version : 0.00*)
(*File Version : 3.23*)

ACTION HMI_PAM_3_Init :
        HMI_PAM_3._000 := 80;
        HMI_PAM_3._010 := 8000;
        HMI_PAM_3._100 := 2500;
        HMI_PAM_3._101 := 2500;
        HMI_PAM_3._102 := 0;
        HMI_PAM_3._103 := 0;
        HMI_PAM_3._104 := 0;
        HMI_PAM_3._105 := 0;
        HMI_PAM_3._106 := 0;
        HMI_PAM_3._107 := 0;
        HMI_PAM_3._108 := 0;
        HMI_PAM_3._109 := 0;
        HMI_PAM_3._112 := 0;
        HMI_PAM_3._113 := 0;
        HMI_PAM_3._200 := 80;
        HMI_PAM_3._210 := 8000;
        HMI_PAM_3._400 := 4;
        HMI_PAM_3._401 := 4;
        HMI_PAM_3._410 := 0;
        HMI_PAM_3._500 := 3;
        HMI_PAM_3._501 := 5;
        HMI_PAM_3._502 := 3;
        HMI_PAM_3._503 := 20;
        HMI_PAM_3._504 := 50000;
        HMI_PAM_3._505 := 10;
        HMI_PAM_3._506 := 3;
        HMI_PAM_3._507 := 5;
        HMI_PAM_3._508 := 3;
        HMI_PAM_3._510 := 1;
        HMI_PAM_3._511 := 19295;
        HMI_PAM_3._512 := 131976;
        HMI_PAM_3._513 := 3;
        HMI_PAM_3._520 := 100;
        HMI_PAM_3._521 := 100;
        HMI_PAM_3._525 := 3;
        HMI_PAM_3._526 := 300;
        HMI_PAM_3._527 := 1;
        HMI_PAM_3._528 := 0;
        HMI_PAM_3._529 := 1800;
        HMI_PAM_3._530 := 3;
        HMI_PAM_3._531 := 300;
        HMI_PAM_3._532 := 1;
        HMI_PAM_3._534 := 1800;
        HMI_PAM_3._540 := 0;
        HMI_PAM_3._550 := 0;
        HMI_PAM_3._551 := 100;
        HMI_PAM_3._554 := 0;
        HMI_PAM_3._555 := 100;
        HMI_PAM_3._558 := 0;
        HMI_PAM_3._559 := 100;
        HMI_PAM_3._562 := 0;
        HMI_PAM_3._563 := 100;
        HMI_PAM_3._566 := 0;
        HMI_PAM_3._567 := 60;
        HMI_PAM_3._570 := 0;
        HMI_PAM_3._571 := 65;
        HMI_PAM_3._572 := 0;
        HMI_PAM_3._573 := 65;
        HMI_PAM_3._574 := 0;
        HMI_PAM_3._575 := 65;
        HMI_PAM_3._600 := 0;
        HMI_PAM_3._601 := 0;
        HMI_PAM_3._602 := 0;
        HMI_PAM_3._603 := 0;
        HMI_PAM_3._604 := 0;
        HMI_PAM_3._605 := 0;
        HMI_PAM_3._606 := 0;
        HMI_PAM_3._607 := 0;
        HMI_PAM_3._608 := 0;
        HMI_PAM_3._609 := 0;
        HMI_PAM_3._610 := 0;
        HMI_PAM_3._611 := 10;
        HMI_PAM_3._612 := 10;
        HMI_PAM_3._613 := 10;
        HMI_PAM_3._614 := 10;
        HMI_PAM_3._615 := 0;
        HMI_PAM_3._616 := 20;
        HMI_PAM_3._620 := 0;
        HMI_PAM_3._621 := 0;
        HMI_PAM_3._622 := 0;
        HMI_PAM_3._623 := 0;
        HMI_PAM_3._624 := 0;
        HMI_PAM_3._625 := 0;
        HMI_PAM_3._626 := 0;
        HMI_PAM_3._627 := 0;
        HMI_PAM_3._628 := 0;
        HMI_PAM_3._629 := 0;
        HMI_PAM_3._630 := 0;
        HMI_PAM_3._631 := 0;
        HMI_PAM_3._632 := 0;
        HMI_PAM_3._633 := 0;
        HMI_PAM_3._634 := 10;
        HMI_PAM_3._635 := 10;
        HMI_PAM_3._636 := 10;
        HMI_PAM_3._637 := 10;
        HMI_PAM_3._640 := 0;
        HMI_PAM_3._641 := 0;
        HMI_PAM_3._642 := 0;
        HMI_PAM_3._643 := 0;
        HMI_PAM_3._644 := 0;
        HMI_PAM_3._645 := 0;
END_ACTION
```

#### HMI_PAM_A1.st
```iecst
(*HMI_PAM_A1 Initialization Action for Filler PLC*)
(*Author = ????*)
(*DB Version : 0.00*)
(*File Version : 3,17*)

ACTION HMI_PAM_A1_Init :
        HMI_PAM_A1._000 := 0;
        HMI_PAM_A1._001 := 0;
        HMI_PAM_A1._002 := 0;
        HMI_PAM_A1._005 := 0;
        HMI_PAM_A1._006 := 0;
        HMI_PAM_A1._007 := 0;
        HMI_PAM_A1._010 := 0;
        HMI_PAM_A1._011 := 0;
        HMI_PAM_A1._012 := 0;
        HMI_PAM_A1._015 := 0;
        HMI_PAM_A1._016 := 0;
        HMI_PAM_A1._017 := 0;
        HMI_PAM_A1._020 := 0;
        HMI_PAM_A1._021 := 0;
        HMI_PAM_A1._022 := 0;
        HMI_PAM_A1._025 := 0;
        HMI_PAM_A1._026 := 0;
        HMI_PAM_A1._027 := 0;
        HMI_PAM_A1._030 := 0;
        HMI_PAM_A1._031 := 0;
        HMI_PAM_A1._032 := 0;
        HMI_PAM_A1._035 := 0;
        HMI_PAM_A1._036 := 0;
        HMI_PAM_A1._037 := 0;
        HMI_PAM_A1._040 := 0;
        HMI_PAM_A1._041 := 0;
        HMI_PAM_A1._042 := 0;
        HMI_PAM_A1._045 := 0;
        HMI_PAM_A1._046 := 0;
        HMI_PAM_A1._047 := 0;
        HMI_PAM_A1._050 := 0;
        HMI_PAM_A1._051 := 0;
        HMI_PAM_A1._052 := 0;
        HMI_PAM_A1._055 := 0;
        HMI_PAM_A1._056 := 0;
        HMI_PAM_A1._057 := 0;
        HMI_PAM_A1._060 := 0;
        HMI_PAM_A1._061 := 0;
        HMI_PAM_A1._062 := 0;
        HMI_PAM_A1._400 := 0;
        HMI_PAM_A1._401 := 0;
        HMI_PAM_A1._402 := 0;
END_ACTION
```

#### HMI_PAM_B1.st
```iecst
(*HMI_PAM_B1 Initialization Action for Filler PLC*)
(*Author = ????*)
(*DB Version : 0.00*)
(*File Version : 3,17*)

ACTION HMI_PAM_B1_Init :
        HMI_PAM_B1._000 := 0;
        HMI_PAM_B1._001 := 40;
        HMI_PAM_B1._005 := 1;
        HMI_PAM_B1._006 := 40;
        HMI_PAM_B1._010 := 0;
        HMI_PAM_B1._011 := 40;
        HMI_PAM_B1._015 := 1;
        HMI_PAM_B1._016 := 40;
        HMI_PAM_B1._020 := 0;
        HMI_PAM_B1._021 := 40;
        HMI_PAM_B1._025 := 1;
        HMI_PAM_B1._026 := 40;
        HMI_PAM_B1._030 := 0;
        HMI_PAM_B1._031 := 40;
        HMI_PAM_B1._035 := 1;
        HMI_PAM_B1._036 := 40;
        HMI_PAM_B1._040 := 0;
        HMI_PAM_B1._041 := 40;
        HMI_PAM_B1._045 := 1;
        HMI_PAM_B1._046 := 40;
        HMI_PAM_B1._050 := 1;
        HMI_PAM_B1._051 := 40;
        HMI_PAM_B1._500 := 5;
        HMI_PAM_B1._501 := 60;
        HMI_PAM_B1._505 := 0;
        HMI_PAM_B1._506 := 100;
        HMI_PAM_B1._510 := 0;
        HMI_PAM_B1._511 := 100;
        HMI_PAM_B1._515 := 0;
        HMI_PAM_B1._516 := 100;
        HMI_PAM_B1._520 := 0;
        HMI_PAM_B1._521 := 100;
        HMI_PAM_B1._525 := 0;
        HMI_PAM_B1._526 := 100;
        HMI_PAM_B1._530 := 0;
        HMI_PAM_B1._531 := 100;
        HMI_PAM_B1._535 := 0;
        HMI_PAM_B1._536 := 100;
        HMI_PAM_B1._540 := 0;
        HMI_PAM_B1._541 := 100;
        HMI_PAM_B1._545 := 0;
        HMI_PAM_B1._546 := 100;
END_ACTION
```

#### HMI_PAM_C1.st
```iecst
(*HMI_PAM_C1 Initialization Action for Filler PLC*)
(*Author = ????*)
(*DB Version : 0.00*)
(*File Version : 3,17*)

ACTION HMI_PAM_C1_Init :
        HMI_PAM_C1._000 := 0;
        HMI_PAM_C1._001 := 0;
        HMI_PAM_C1._002 := 0;
        HMI_PAM_C1._003 := 0;
        HMI_PAM_C1._004 := 0;
        HMI_PAM_C1._005 := 0;
        HMI_PAM_C1._006 := 0;
        HMI_PAM_C1._007 := 0;
        HMI_PAM_C1._008 := 0;
        HMI_PAM_C1._009 := 0;
        HMI_PAM_C1._010 := 0;
        HMI_PAM_C1._011 := 0;
        HMI_PAM_C1._012 := 0;
        HMI_PAM_C1._013 := 0;
        HMI_PAM_C1._014 := 0;
        HMI_PAM_C1._015 := 0;
        HMI_PAM_C1._016 := 0;
        HMI_PAM_C1._017 := 0;
        HMI_PAM_C1._018 := 0;
        HMI_PAM_C1._019 := 0;
        HMI_PAM_C1._020 := 0;
        HMI_PAM_C1._021 := 0;
        HMI_PAM_C1._022 := 0;
        HMI_PAM_C1._023 := 0;
        HMI_PAM_C1._024 := 0;
        HMI_PAM_C1._025 := 0;
        HMI_PAM_C1._026 := 0;
        HMI_PAM_C1._027 := 0;
        HMI_PAM_C1._028 := 0;
        HMI_PAM_C1._029 := 0;
        HMI_PAM_C1._030 := 0;
        HMI_PAM_C1._031 := 0;
        HMI_PAM_C1._032 := 0;
        HMI_PAM_C1._033 := 0;
        HMI_PAM_C1._034 := 0;
        HMI_PAM_C1._035 := 0;
        HMI_PAM_C1._036 := 0;
        HMI_PAM_C1._037 := 0;
        HMI_PAM_C1._038 := 0;
        HMI_PAM_C1._039 := 0;
        HMI_PAM_C1._040 := 0;
        HMI_PAM_C1._041 := 0;
        HMI_PAM_C1._042 := 0;
        HMI_PAM_C1._043 := 0;
        HMI_PAM_C1._044 := 0;
        HMI_PAM_C1._045 := 0;
        HMI_PAM_C1._046 := 0;
        HMI_PAM_C1._047 := 0;
        HMI_PAM_C1._048 := 0;
        HMI_PAM_C1._049 := 0;
        HMI_PAM_C1._050 := 0;
        HMI_PAM_C1._051 := 0;
        HMI_PAM_C1._052 := 0;
        HMI_PAM_C1._053 := 0;
        HMI_PAM_C1._054 := 0;
        HMI_PAM_C1._055 := 0;
        HMI_PAM_C1._056 := 0;
        HMI_PAM_C1._057 := 0;
        HMI_PAM_C1._058 := 0;
        HMI_PAM_C1._059 := 0;
        HMI_PAM_C1._060 := 0;
        HMI_PAM_C1._061 := 0;
        HMI_PAM_C1._062 := 0;
        HMI_PAM_C1._063 := 0;
        HMI_PAM_C1._064 := 0;
        HMI_PAM_C1._065 := 0;
        HMI_PAM_C1._066 := 0;
        HMI_PAM_C1._067 := 0;
        HMI_PAM_C1._068 := 0;
        HMI_PAM_C1._069 := 0;
        HMI_PAM_C1._070 := 0;
        HMI_PAM_C1._071 := 0;
        HMI_PAM_C1._072 := 0;
        HMI_PAM_C1._073 := 0;
        HMI_PAM_C1._074 := 0;
        HMI_PAM_C1._075 := 0;
        HMI_PAM_C1._076 := 0;
        HMI_PAM_C1._077 := 0;
        HMI_PAM_C1._078 := 0;
        HMI_PAM_C1._079 := 0;
        HMI_PAM_C1._080 := 0;
        HMI_PAM_C1._081 := 0;
        HMI_PAM_C1._082 := 0;
        HMI_PAM_C1._083 := 0;
        HMI_PAM_C1._084 := 0;
        HMI_PAM_C1._085 := 0;
        HMI_PAM_C1._086 := 0;
        HMI_PAM_C1._087 := 0;
        HMI_PAM_C1._088 := 0;
        HMI_PAM_C1._089 := 0;
        HMI_PAM_C1._090 := 0;
        HMI_PAM_C1._091 := 0;
        HMI_PAM_C1._092 := 0;
        HMI_PAM_C1._093 := 0;
        HMI_PAM_C1._094 := 0;
        HMI_PAM_C1._095 := 0;
        HMI_PAM_C1._096 := 0;
        HMI_PAM_C1._097 := 0;
        HMI_PAM_C1._098 := 0;
        HMI_PAM_C1._099 := 0;
        HMI_PAM_C1._100 := 0;
        HMI_PAM_C1._101 := 0;
        HMI_PAM_C1._102 := 0;
        HMI_PAM_C1._103 := 0;
        HMI_PAM_C1._104 := 0;
        HMI_PAM_C1._105 := 0;
        HMI_PAM_C1._106 := 0;
        HMI_PAM_C1._107 := 0;
        HMI_PAM_C1._108 := 0;
        HMI_PAM_C1._109 := 0;
        HMI_PAM_C1._110 := 0;
        HMI_PAM_C1._111 := 0;
        HMI_PAM_C1._112 := 0;
        HMI_PAM_C1._113 := 0;
        HMI_PAM_C1._114 := 0;
        HMI_PAM_C1._115 := 0;
        HMI_PAM_C1._116 := 0;
        HMI_PAM_C1._117 := 0;
        HMI_PAM_C1._118 := 0;
        HMI_PAM_C1._119 := 0;
END_ACTION
```

#### HMI_PAM_D1.st
```iecst
(*HMI_PAM_D1 Initialization Action for Filler PLC*)
(*Author = ????*)
(*DB Version : 0.00*)
(*File Version : 3,17*)

ACTION HMI_PAM_D1_Init :
        HMI_PAM_D1._000 := 0;
        HMI_PAM_D1._001 := 0;
        HMI_PAM_D1._002 := 0;
        HMI_PAM_D1._003 := 0;
        HMI_PAM_D1._004 := 0;
        HMI_PAM_D1._005 := 0.5;
        HMI_PAM_D1._006 := 1;
        HMI_PAM_D1._007 := 0;
        HMI_PAM_D1._008 := 0;
        HMI_PAM_D1._009 := 0;
        HMI_PAM_D1._010 := 0;
        HMI_PAM_D1._011 := 0;
        HMI_PAM_D1._012 := 0;
        HMI_PAM_D1._013 := 0;
        HMI_PAM_D1._014 := 0;
        HMI_PAM_D1._015 := 0;
        HMI_PAM_D1._016 := 0;
        HMI_PAM_D1._017 := 0;
        HMI_PAM_D1._018 := 0;
        HMI_PAM_D1._019 := 0;
        HMI_PAM_D1._020 := 0;
        HMI_PAM_D1._021 := 0;
        HMI_PAM_D1._022 := 0;
        HMI_PAM_D1._023 := 0;
        HMI_PAM_D1._024 := 0;
        HMI_PAM_D1._025 := 0;
        HMI_PAM_D1._026 := 0;
        HMI_PAM_D1._027 := 0;
        HMI_PAM_D1._028 := 0;
        HMI_PAM_D1._029 := 0;
        HMI_PAM_D1._030 := 0;
        HMI_PAM_D1._031 := 0;
        HMI_PAM_D1._032 := 0;
        HMI_PAM_D1._033 := 0;
        HMI_PAM_D1._034 := 0;
        HMI_PAM_D1._035 := 0;
        HMI_PAM_D1._036 := 0;
        HMI_PAM_D1._037 := 0;
        HMI_PAM_D1._038 := 0;
        HMI_PAM_D1._039 := 0;
        HMI_PAM_D1._040 := 0;
        HMI_PAM_D1._041 := 0;
        HMI_PAM_D1._042 := 0;
        HMI_PAM_D1._043 := 0;
        HMI_PAM_D1._044 := 0;
        HMI_PAM_D1._045 := 0;
        HMI_PAM_D1._046 := 0;
        HMI_PAM_D1._047 := 0;
        HMI_PAM_D1._048 := 0;
        HMI_PAM_D1._049 := 0;
        HMI_PAM_D1._050 := 0;
        HMI_PAM_D1._051 := 0;
        HMI_PAM_D1._052 := 0;
        HMI_PAM_D1._053 := 0;
        HMI_PAM_D1._054 := 0;
        HMI_PAM_D1._055 := 0;
        HMI_PAM_D1._056 := 0;
        HMI_PAM_D1._057 := 0;
        HMI_PAM_D1._058 := 0;
        HMI_PAM_D1._059 := 0;
        HMI_PAM_D1._060 := 0;
        HMI_PAM_D1._061 := 0;
        HMI_PAM_D1._062 := 0;
        HMI_PAM_D1._063 := 0;
        HMI_PAM_D1._064 := 0;
        HMI_PAM_D1._065 := 0;
        HMI_PAM_D1._066 := 0;
        HMI_PAM_D1._067 := 0;
        HMI_PAM_D1._068 := 0;
        HMI_PAM_D1._069 := 0;
        HMI_PAM_D1._070 := 0;
        HMI_PAM_D1._071 := 0;
        HMI_PAM_D1._072 := 0;
        HMI_PAM_D1._073 := 0;
        HMI_PAM_D1._074 := 0;
        HMI_PAM_D1._075 := 0;
        HMI_PAM_D1._076 := 0;
        HMI_PAM_D1._077 := 0;
        HMI_PAM_D1._078 := 0;
        HMI_PAM_D1._079 := 0;
        HMI_PAM_D1._080 := 0;
        HMI_PAM_D1._081 := 0;
        HMI_PAM_D1._082 := 0;
        HMI_PAM_D1._083 := 0;
        HMI_PAM_D1._084 := 0;
        HMI_PAM_D1._085 := 0;
        HMI_PAM_D1._086 := 0;
        HMI_PAM_D1._087 := 0;
        HMI_PAM_D1._088 := 0;
        HMI_PAM_D1._089 := 0;
        HMI_PAM_D1._090 := 10;
        HMI_PAM_D1._091 := 10;
        HMI_PAM_D1._092 := 1;
        HMI_PAM_D1._093 := 0;
        HMI_PAM_D1._094 := 0;
        HMI_PAM_D1._095 := 0.7;
        HMI_PAM_D1._096 := 1;
        HMI_PAM_D1._097 := 1;
        HMI_PAM_D1._098 := 0;
        HMI_PAM_D1._099 := 0;
        HMI_PAM_D1._500 := 0;
        HMI_PAM_D1._501 := 40;
        HMI_PAM_D1._502 := 0;
        HMI_PAM_D1._503 := 0;
        HMI_PAM_D1._504 := 0;
        HMI_PAM_D1._505 := 1.5;
        HMI_PAM_D1._506 := 0.6;
        HMI_PAM_D1._507 := 0;
        HMI_PAM_D1._508 := 0;
        HMI_PAM_D1._509 := 0;
        HMI_PAM_D1._510 := 0;
        HMI_PAM_D1._511 := 0;
        HMI_PAM_D1._512 := 0;
        HMI_PAM_D1._513 := 0;
        HMI_PAM_D1._514 := 0;
        HMI_PAM_D1._515 := 0;
        HMI_PAM_D1._516 := 0;
        HMI_PAM_D1._517 := 0;
        HMI_PAM_D1._518 := 0;
        HMI_PAM_D1._519 := 0;
        HMI_PAM_D1._520 := 0;
        HMI_PAM_D1._521 := 0;
        HMI_PAM_D1._522 := 0;
        HMI_PAM_D1._523 := 0;
        HMI_PAM_D1._524 := 0;
        HMI_PAM_D1._525 := 0;
        HMI_PAM_D1._526 := 0;
        HMI_PAM_D1._527 := 0;
        HMI_PAM_D1._528 := 0;
        HMI_PAM_D1._529 := 0;
        HMI_PAM_D1._530 := 0;
        HMI_PAM_D1._531 := 0;
        HMI_PAM_D1._532 := 0;
        HMI_PAM_D1._533 := 0;
        HMI_PAM_D1._534 := 0;
        HMI_PAM_D1._535 := 0;
        HMI_PAM_D1._536 := 0;
        HMI_PAM_D1._537 := 0;
        HMI_PAM_D1._538 := 0;
        HMI_PAM_D1._539 := 0;
        HMI_PAM_D1._540 := 0;
        HMI_PAM_D1._541 := 0;
        HMI_PAM_D1._542 := 0;
        HMI_PAM_D1._543 := 0;
        HMI_PAM_D1._544 := 0;
        HMI_PAM_D1._545 := 0;
        HMI_PAM_D1._546 := 0;
        HMI_PAM_D1._547 := 0;
        HMI_PAM_D1._548 := 0;
        HMI_PAM_D1._549 := 0;
        HMI_PAM_D1._550 := 0;
        HMI_PAM_D1._551 := 0;
        HMI_PAM_D1._552 := 0;
        HMI_PAM_D1._553 := 0;
        HMI_PAM_D1._554 := 0;
        HMI_PAM_D1._555 := 0;
        HMI_PAM_D1._556 := 0;
        HMI_PAM_D1._557 := 0;
        HMI_PAM_D1._558 := 0;
        HMI_PAM_D1._559 := 0;
        HMI_PAM_D1._560 := 0;
        HMI_PAM_D1._561 := 0;
        HMI_PAM_D1._562 := 0;
        HMI_PAM_D1._563 := 0;
        HMI_PAM_D1._564 := 0;
        HMI_PAM_D1._565 := 0;
        HMI_PAM_D1._566 := 0;
        HMI_PAM_D1._567 := 0;
        HMI_PAM_D1._568 := 0;
        HMI_PAM_D1._569 := 0;
        HMI_PAM_D1._570 := 0;
        HMI_PAM_D1._571 := 0;
        HMI_PAM_D1._572 := 0;
        HMI_PAM_D1._573 := 0;
        HMI_PAM_D1._574 := 0;
        HMI_PAM_D1._575 := 0;
        HMI_PAM_D1._576 := 0;
        HMI_PAM_D1._577 := 0;
        HMI_PAM_D1._578 := 0;
        HMI_PAM_D1._579 := 0;
        HMI_PAM_D1._580 := 0;
        HMI_PAM_D1._581 := 0;
        HMI_PAM_D1._582 := 0;
        HMI_PAM_D1._583 := 0;
        HMI_PAM_D1._584 := 0;
        HMI_PAM_D1._585 := 0;
        HMI_PAM_D1._586 := 0;
        HMI_PAM_D1._587 := 0;
        HMI_PAM_D1._588 := 0;
        HMI_PAM_D1._589 := 0;
        HMI_PAM_D1._590 := 0;
        HMI_PAM_D1._591 := 0;
        HMI_PAM_D1._592 := 0;
        HMI_PAM_D1._593 := 0;
        HMI_PAM_D1._594 := 0;
        HMI_PAM_D1._595 := 0;
        HMI_PAM_D1._596 := 0;
        HMI_PAM_D1._597 := 0;
        HMI_PAM_D1._598 := 0;
        HMI_PAM_D1._599 := 0;
        HMI_PAM_D1._611 := 0;
        HMI_PAM_D1._612 := 0;
        HMI_PAM_D1._613 := 0;
        HMI_PAM_D1._614 := 0;
        HMI_PAM_D1._615 := 0;
        HMI_PAM_D1._616 := 0;
        HMI_PAM_D1._617 := 0;
        HMI_PAM_D1._618 := 0;
        HMI_PAM_D1._619 := 0;
        HMI_PAM_D1._620 := 0;
END_ACTION
```

#### HMI_PAT_1.st
```iecst
(*HMI_PAT_1 Initialization Action for Filler PLC*)
(*Author = ????*)
(*DB Version : 0.00*)
(*File Version : 3,17*)

ACTION HMI_PAT_1_Init :
        HMI_PAT_1._010 := 0;
        HMI_PAT_1._011 := 0;
        HMI_PAT_1._100 := 150;
        HMI_PAT_1._101 := 200;
        HMI_PAT_1._110 := 20;
        HMI_PAT_1._420 := 450;
        HMI_PAT_1._421 := 1000;
        HMI_PAT_1._422 := 200;
        HMI_PAT_1._423 := 7200;
        HMI_PAT_1._424 := 1800;
        HMI_PAT_1._425 := 20;
        HMI_PAT_1._426 := 600;
END_ACTION
```

#### Variable.var
```iecst
VAR
	TMR_TON_ParInitialization : TON;
	VAR_PAR_Initialization : BOOL;
END_VAR
```

### PAR.var - Global variables
```iecst
(*MACHINE PARAMETERS*)
VAR RETAIN
	HMI_PAM_1 : HMI_PAM_1_Type;
END_VAR
VAR
	HMI_CFG_PAM_1 : PAM_CFG_Type;
END_VAR
VAR RETAIN
	HMI_PAM_3 : HMI_PAM_3_Type;
END_VAR
VAR
	HMI_CFG_PAM_3 : PAM_CFG_Type;
END_VAR
VAR RETAIN
	HMI_PAM_A1 : HMI_PAM_A1_Type;
END_VAR
VAR
	HMI_CFG_PAM_A1 : PAM_CFG_Type;
END_VAR
VAR RETAIN
	HMI_PAM_B1 : HMI_PAM_B1_Type;
END_VAR
VAR
	HMI_CFG_PAM_B1 : PAM_CFG_Type;
END_VAR
VAR RETAIN
	HMI_PAM_C1 : HMI_PAM_C1_Type;
END_VAR
VAR
	HMI_CFG_PAM_C1 : PAM_CFG_Type;
END_VAR
VAR RETAIN
	HMI_PAM_D1 : HMI_PAM_D1_Type;
END_VAR
VAR
	HMI_CFG_PAM_D1 : PAM_CFG_Type;
END_VAR
(*MACHINE RECIPE PARAMETERS*)
VAR RETAIN
	HMI_PAR_1 : HMI_PAR_1_Type;
END_VAR
VAR
	HMI_CFG_PAR_1 : PAR_CFG_Type;
END_VAR
(*MACHINE TECNOLOGICAL PARAMETERS*)
VAR RETAIN
	HMI_PAT_1 : HMI_PAT_1_Type;
END_VAR
VAR
	HMI_CFG_PAT_1 : PAM_CFG_Type;
END_VAR
(*MACHINE CONFIGURATION PARAMETERS*)
VAR RETAIN
	HMI_PAC_1 : HMI_PAC_1_Type;
END_VAR
VAR
	HMI_CFG_PAC_1 : PAM_CFG_Type;
END_VAR
(*MACHINE OPTION PARAMETERS*)
VAR
	HMI_PAO_2 : HMI_PAO_2_Type;
END_VAR
```
